REGION Network 4: Block description — Section 3.3 to 3.5
   // ▂▂▂▂▂▂▂▂▂▂▂▂▂▂▂▂▂▂▂▂▂▂▂▂▂▂▂▂▂▂▂▂▂▂▂▂▂▂▂▂▂▂▂▂
   // 3.3     Fault handling
   // 
   // 
   // There are five fault conditions, four are derived from position faults and one from an external 
   // fault signal:
   // 
   //  ――――――――――――――――――――――――――――――――――――――――――
   //  FAULT         DESCRIPTION                     LATCHING
   //  ――――――――――――――――――――――――――――――――――――――――――
   //  Failed to open      Valve failed to open in the specified               YES
   //             opening operation time
   // 
   //  Failed to close      Valve failed to close in the specified              YES
   //             closing operation time
   // 
   //  Failed while open   Valve suffered position failure while            YES
   //             in a static OPEN state
   // 
   //  Failed while closed   Valve suffered position failure while            YES
   //             in a static CLOSED state
   // 
   //  External fault        The EXT_FAULT signal is active                 NO
   //   ――――――――――――――――――――――――――――――――――――――――――
   // 
   // If any of the above faults are active, the valve will be deenergised (both the OPEN_CMD and 
   // CLOSE_CMD parameters will be set to 0) and the module will ignore all commands either 
   // automatic or manual and will ignore all interlock conditions.
   // 
   // Note:    If the maintain output option is activated (CONFIG_MAINT_OP = 1), the outputs will be 
   //      deenergised if a fault is present (both the OPEN_CMD and CLOSE_CMD parameters 
   //      will be set to 0).
   // 
   // 
   // 
   // ▁▁▁▁▁▁▁▁▁▁▁▁▁▁▁▁▁▁▁▁▁▁▁▁▁▁▁▁▁▁▁▁▁▁▁▁▁▁▁▁▁▁▁▁
   // 3.3.1    Position faults
   // 
   // 
   // All position faults (derived from position feedback signals) are latching fault conditions that  
   // require the operator to issue a reset command, this is usually via a faceplate available at the 
   // supervisory system (SCADA/HMI), but could also be via a hardwired 
   // (pushbutton) signal. 
   // 
   // The reset signal is specified within the DYNAMIC_DATA parameter UDT as follows:        
   // 
   //  DATA STRUCTURE    UT31101_Dy_DevValveBi
   //  ――――――――――――――――――――――――――――――――――――――――――
   //  SIGNAL         FUNCTION                TYPE     DETAILS
   //  ――――――――――――――――――――――――――――――――――――――――――
   //  mode_Reset        A reset pulse                Bool     1 = reset latched faults
   //            (active for one Controller cycle)            0 = no action
   //  ――――――――――――――――――――――――――――――――――――――――――
   // 
   // 
   // 
   // ▁▁▁▁▁▁▁▁▁▁▁▁▁▁▁▁▁▁▁▁▁▁▁▁▁▁▁▁▁▁▁▁▁▁▁▁▁▁▁▁▁▁▁▁
   // 3.3.2    Resetting position faults
   // 
   // 
   // If a position fault has occurred, and the fault is then reset, the appropriate opening or closing 
   // operation timer will be retriggered, allowing the valve time to achieve the required position.
   // 
   // 
   // 
   // ▁▁▁▁▁▁▁▁▁▁▁▁▁▁▁▁▁▁▁▁▁▁▁▁▁▁▁▁▁▁▁▁▁▁▁▁▁▁▁▁▁▁▁▁
   // 3.3.3    External fault
   // 
   // 
   // The external fault is an optional hardwired signal from the valve, it indicates that the device 
   // itself is registering that there is some problem. Such external fault signals are more commonly 
   // associated with motorised valves (equipped with thermal overload detectors), but may also be 
   // associated with pneumatic or hydraulic operated valves to indicate that the is a 
   // pneumatic/hydraulic system failure.
   // 
   // Such fault signals are generally indicated via a hardwired digital input to the Controller.
   // 
   // The external fault signal (if used) is passed to the module as the parameter: EXT_FAULT .
   // 
   // Any signal connected to the EXT_FAULT parameter must be active high (i.e. the signal must be 
   // set to 1 to indicate the fault condition is present). 
   // 
   // Where a failsafe response signal is used (active when set to 0) is used, it must be inverted at the 
   // EXT_FAULT parameter:
   // 
   // 
   //                         ┌─────────────
   //      ───────────────────┤ FC11101 
   //                         ├───────────────┤
   //           "V001_FAULT"               │               │
   //        ────┤╱├──────────┤ EXT_FAULT             │
   //                         │               
   //                         │               
   // 
   // 
   // If the EXT_FAULT signal is not required, the input should be set to _False  (similar to the safety 
   // and interlock signals that are not used, see § 3.4).
   // 
   // The EXT_FAULT signal is non-latching; it does not require a mode_Reset signal to clear the fault. 
   // The external fault will automatically reset whenever the EXT_FAULT signal is set to 0.
   // 
   // 
   // 
   // ▂▂▂▂▂▂▂▂▂▂▂▂▂▂▂▂▂▂▂▂▂▂▂▂▂▂▂▂▂▂▂▂▂▂▂▂▂▂▂▂▂▂▂▂
   // 3.4     Safety and interlocks
   // 
   // 
   // Safety and interlock signals are optional signals, passed as individual parameters to the module 
   // (in the same a manner as IO signals), all such signals are optional, a valve can have all, none or 
   // any combination of the signals.
   // 
   // Safety and interlock signals all act to override the normal operation of the valve (whether in 
   // automatic or manual mode) and force the valve to a particular state.
   // 
   // There is one safety signal and three interlock signals, each having its own formal module 
   // parameter:
   // 
   // 
   //  SAFETY SIGNAL
   //  ――――――――――――――――――――――――――――――――――――――――――
   //  PARAM        FUNCTION                   TYPE     DETAILS 
   //  ――――――――――――――――――――――――――――――――――――――――――
   //  E_STOP       Safety or emergency stop signals are         Bool     1 = E-stop active
   //          hardwired signals that remove power            0 = healthy
   //          required, set permanently to _False
   //  ――――――――――――――――――――――――――――――――――――――――――
   //  INTERLOCK SIGNALS
   //  ――――――――――――――――――――――――――――――――――――――――――
   //  PARAM        FUNCTION                   TYPE     DETAILS  
   //  ――――――――――――――――――――――――――――――――――――――――――
   //  TRIP       A latching interlock, it activates whenever a      Bool     1 = Trip active
   //          set of events are true and forces the devices        0 = healthy
   //          to a given state. It will not deactivate until the 
   //          triggering conditions are removed and a 
   //          reset signal has been given.
   // 
   //  INTERLOCK    A simple interlock that is active whenever a   Bool     1 = Interlock active
   //          set of conditions is true, it will force the            0 = healthy
   //          devices to a given state
   // 
   //  PERMISSIVE     Takes no action if a device is in a non-        Bool     1 = Permissive active
   //          permitted state, but once the device is in           0 = healthy
   //          that state will prevent a transition back to 
   //          the non-permitted state.
   //  ――――――――――――――――――――――――――――――――――――――――――
   // 
   // 
   // Each safety and interlock signal has its own configuration signal that must be used to formally 
   // disable the parameter if the signal is not required, these are all within the STATIC_DATA parameter 
   // UDT (UT11101_St_DevValveBi) as follows:
   // 
   // 
   //  DATA STRUCTURE    UT11101_St_DevValveBi
   //  ――――――――――――――――――――――――――――――――――――――――――
   //  SIGNAL        FUNCTION              TYPE     DETAILS
   //  ――――――――――――――――――――――――――――――――――――――――――
   //  CONFIG_ESTOP_DIS    Disables the safety signal.        Bool     1 = E_STOP disabled
   //              If set to 1, any signal on the          0 = E_STOP enabled
   //              E_STOP parameter will be 
   //              ignored.
   // 
   //  CONFIG_TRIP_DIS      Disables the trip interlock signal.   Bool     1 = TRIP disabled
   //              If set to 1, any signal on the          0 = TRIP enabled
   //              TRIP parameter will be 
   //              ignored.
   // 
   //  CONFIG_ILOCK_DIS     Disables the interlock signal.    Bool     1 = INTERLOCK disabled
   //              If set to 1, any signal on the          0 = INTERLOCK enabled
   //              INTERLOCK parameter will be 
   //              ignored.
   // 
   //  CONFIG_PERM_DIS   Disables the permissive interlock  Bool     1 = PERMISSIVE disabled
   //              signal. If set to 1, any signal on the       0 = PERMISSIVE enabled
   //              TRIP parameter will be 
   //              ignored.
   //  ――――――――――――――――――――――――――――――――――――――――――
   // 
   // The disable signals are used to formally configure the valve, they allow any supervisory system to 
   // know the correct configuration of the valve and display information accordingly.
   // 
   // 
   // 
   // ▁▁▁▁▁▁▁▁▁▁▁▁▁▁▁▁▁▁▁▁▁▁▁▁▁▁▁▁▁▁▁▁▁▁▁▁▁▁▁▁▁▁▁▁
   // 3.4.1    Safety signal operation
   // 
   // 
   // Safety or emergency stop signals are hardwired signals that remove power from a device forcing 
   // it to a safe state. Such signals act independently of the software (the pressing of an emergency 
   // stop button will physically remove power from the affected devices).
   // 
   // The emergency stop signal is passed to the module as the parameter E_STOP; it informs the 
   // module that the safety signal has been activated and allows the module to adjust the state of 
   // the valve to follow the emergency stop conditions.
   // 
   // When the emergency stop signal is removed, the valve will resume the requested state (with the 
   // appropriate operation timer).
   // 
   // Under emergency stop conditions the valve is always deenergised (both physically by the 
   // hardware and within the software via the actions of this module), both the OPEN_CMD and 
   // CLOSE_CMD outputs set to zero (OPEN_CMD = 0 and CLOSE_CMD = 0).
   // 
   // The emergency stop signal is absolute and will override any other demand made of the valve. 
   // There is no mechanism for bypassing this form of safety signal.
   // 
   // 
   // 
   // ▁▁▁▁▁▁▁▁▁▁▁▁▁▁▁▁▁▁▁▁▁▁▁▁▁▁▁▁▁▁▁▁▁▁▁▁▁▁▁▁▁▁▁▁
   // Safety signal operation when valve is changing state (recovery time)
   // 
   // 
   // In the case of a bistable valve, the removing of the power under emergency stop conditions, 
   // simply deenergises both outputs leaving the valve in its current state: if the valve were already 
   // open, it would remain open, similarly if the valve were closed, it would remain closed.
   // 
   // Additionally, if the valve were in the process of changing state (either opening or closing) when 
   // the emergency stop occurred, the same thing happens, both outputs are deenergised and the 
   // valve simply stops where it is in mid-transition (i.e. in some indeterminate, intermediate state 
   // between open and closed). 
   // 
   // To accommodate this condition, the active operation timer will simply pause at its current 
   // elapsed value (the value reached when the emergency stop activated) and the valve will 
   // remain in either the opening or closing state; i.e. status_Opening or status_Closing will remain 
   // active until the emergency stop condition is removed.
   // 
   // Under these conditions (an emergency stop while changing state), the removal of the 
   // emergency stop tiggers a recovery timer, this is used to delay the restarting of the operation 
   // timer (or the run-on timer if it is active), the recover timer is used to allow the physical aspects 
   // of the valve itself to reset and resume operation (e.g. to allow the valve to power-up and the 
   // motor to ramp to the correct speed &c.), this recovery time is configurable.
   // 
   // Note:    The recovery timer will also run when the emergency stop condition is removed 
   //      even if the valve is in a defined position, under these circumstances, the operation 
   //      timer will again be delayed until the recovery timer is complete (this avoids a 
   //      situation where the valve is required to change state immediately after an estop 
   //      while the valve motor is still recovering — again it effectively extends the operation 
   //      timer sufficiently to allow the valve to recover).
   // 
   // The recovery time preset is specified in the STATIC_DATA parameter 
   // UDT (UT11101_St_DevValveBi) as follows. It is the same irrespective of whether the valve was 
   // opening or closing.
   // 
   // 
   //  DATA STRUCTURE    UT11101_St_DevValveBi
   //  ――――――――――――――――――――――――――――――――――――――――――
   //  SIGNAL        FUNCTION              TYPE     DETAILS
   //  ――――――――――――――――――――――――――――――――――――――――――
   //  TIME_RECOVERY       Recovery delay time, delays the     Real     Seconds
   //              restarting of the operation time 
   //              if an E stop occurred while 
   //              changing state
   //  ――――――――――――――――――――――――――――――――――――――――――
   // 
   // 
   // If the recovery timer is active, the elapsed (counting down) time is stored within the 
   // DYNAMIC_DATA parameter UDT (UT31101_Dy_DevValveBi) as follows:
   // 
   // 
   //  DATA STRUCTURE    UT31101_Dy_DevValveBi
   //  ――――――――――――――――――――――――――――――――――――――――――
   //  SIGNAL        FUNCTION              TYPE     DETAILS
   //  ――――――――――――――――――――――――――――――――――――――――――
   //  actual_Recovery_Timer    Actual (elapsed) value of     Real     Seconds
   //              the recovery timer  
   //  ――――――――――――――――――――――――――――――――――――――――――
   // 
   // 
   // Again, the recovery timer counts down from the TIME_RECOVERY value to zero, at which point, the 
   // operation timer will restart from the elapsed time.
   // 
   // Note:    During the recovery period, the appropriate OPEN_CMD or CLOSE_CMD output will 
   //      reactivate (depending on whether the valve was originally opening or closing).
   // 
   // 
   // 
   // ▁▁▁▁▁▁▁▁▁▁▁▁▁▁▁▁▁▁▁▁▁▁▁▁▁▁▁▁▁▁▁▁▁▁▁▁▁▁▁▁▁▁▁▁
   // Typical usage of the E_STOP parameter
   // 
   // 
   // Any safety signal connected to the E_STOP parameter must be active high (i.e. the signal must be 
   // set to 1 to activate the safety signal response). It is often the case, where hardwired emergency 
   // stop signals are used, that the emergency stop condition is activated by the absence of a signal 
   // (a failsafe response) rather than the application of a signal. The module can accommodate this 
   // sense of signal by inverting the E_STOP input:
   // 
   // 
   //                         ┌─────────────
   //      ───────────────────┤ FC11101 
   //                         ├───────────────┤
   //           "ZONEA_ESTOP"              │               │
   //        ────┤╱├──────────┤ E_STOP             │
   //                         │               
   //                         │               
   // 
   // 
   // If no safety signal is used, the parameter is set to the _False tag (note, also that the configuration 
   // signal CONFIG_ESTOP_DIS should also be set to 1):
   // 
   // 
   //                         ┌─────────────
   //      ───────────────────┤ FC11101 
   //                         ├───────────────┤
   //                         │               │
   //                      _False ──┤ E_STOP             │
   //                         │               
   //                         │    
   // 
   // 
   // 
   // ▁▁▁▁▁▁▁▁▁▁▁▁▁▁▁▁▁▁▁▁▁▁▁▁▁▁▁▁▁▁▁▁▁▁▁▁▁▁▁▁▁▁▁▁
   // 3.4.2    Interlock signals
   // 
   // 
   // Interlock signals are a more flexible mechanism for overriding the requested position of the valve. 
   // Interlock signals can be both hardware driven (similar to a safety signal) or can be purely software 
   // derived (unlike a safety signal).
   // 
   // Software derived interlock signals can accommodate more complex and more flexible 
   // arrangements, it would for example, be possible to disable a software derived interlock if the 
   // process were undergoing some particular function, such as cleaning &c.
   // 
   // There are three different types of interlock arrangements:
   // 
   // There are three types of interlock signal:
   // 
   //    1.  INTERLOCK
   //      A simple interlock that is active whenever a set of conditions is true, it will force any 
   //      associated devices to a given safe state.
   // 
   //    2.  PERMISSIVE
   //      Takes no action if a device is in a non-safe state, but once the device is in a safe 
   //      state will prevent a transition to a non-safe state (i.e. will not force a valve to close, 
   //      but once it is closed, will prevent it from re-opening).
   // 
   //    3.  TRIP
   //      A latching interlock, it activates whenever a set of events are true (like an interlock), 
   //      but will not deactivate until the triggering conditions are removed and a reset signal 
   //      has been given (effectively a latching interlock), it will force any associated devices 
   //      to a given safe state.
   // 
   // For any type of interlock, the specified interlock state (or permitted state) can be either open or 
   // closed irrespective of the type of valve (normally open or normally closed); unlike the safety signal, 
   // it does not have to be the deenergised state of the valve.
   // 
   // That said, the most common interlock state is the deenergised state of the valve; i.e. the failsafe 
   // position of the valve.
   // 
   // 
   // 
   // ▁▁▁▁▁▁▁▁▁▁▁▁▁▁▁▁▁▁▁▁▁▁▁▁▁▁▁▁▁▁▁▁▁▁▁▁▁▁▁▁▁▁▁▁
   // Typical usage of interlock signals
   // 
   // 
   // Each type of interlock is passed as its own parameter: TRIP, INTERLOCK or PERMISSIVE. Like the 
   // safety signal (E_STOP), each parameter is active high (i.e. the signal must be set to 1 to activate 
   // the associated interlock signal response). 
   // 
   // Again, it is often the case, where hardwired interlock signals are used, that the condition is 
   // activated by the absence of a signal (i.e. a failsafe response) rather than the application of a 
   // signal. The module can accommodate this sense of signal by inverting the relevant input:
   // 
   // 
   //                         ┌─────────────
   //      ───────────────────┤ FC11101 
   //                         ├───────────────┤
   //        "DB23102_Dy_Perm.V001"     │               │
   //        ────┤╱├──────────┤ PERMISSIVE           │
   //                         │               
   // 
   // If a particular interlock signal is not used, the parameter is set to the _False tag (note also: that 
   // the appropriate configuration signal should also be set to 1: CONFIG_TRIP_DIS, CONFIG_ILOCK_DIS 
   // or CONFIG_PERM_DIS).
   // 
   //                         ┌─────────────
   //      ───────────────────┤ FC11101 
   //                         ├───────────────┤
   //                         │               │
   //                      _False ──┤ TRIP                    │
   //                         │               
   //                         │  
   // 
   // 
   // 
   // ▁▁▁▁▁▁▁▁▁▁▁▁▁▁▁▁▁▁▁▁▁▁▁▁▁▁▁▁▁▁▁▁▁▁▁▁▁▁▁▁▁▁▁▁
   // Configuring the interlock signals
   // 
   // 
   // The state adopted by the valve when a particular interlock is active (TRIP or INTERLOCK) or the 
   // permitted state of the valve (PERMISSIVE) are set individually for each type of interlock signal. 
   // These configuration signals are stored within the STATIC_DATA parameter UDT as follows:
   // 
   // 
   //  DATA STRUCTURE    UT11101_St_DevValveBi
   // 
   //  ――――――――――――――――――――――――――――――――――――――――――
   //  SIGNAL        FUNCTION              TYPE     DETAILS
   //  ――――――――――――――――――――――――――――――――――――――――――
   //  CONFIG_TRIP_OP_CL   The required state of a valve if     Bool     1 = valve will open
   //              the TRIP signal is active            0 = valve will close
   // 
   //  CONFIG_ILOCK_OP_CL  The required state of a valve if     Bool     1 = valve will open
   //              the INTERLOCK signal is active         0 = valve will close
   // 
   //  CONFIG_PERM_OP_CL  The permitted state of a valve if   Bool     1 = valve may open
   //              the PERMISSIVE signal is active          0 = valve may close
   //  ――――――――――――――――――――――――――――――――――――――――――
   // 
   // For example, if CONFIG_ILOCK_OP_CL is set to 1, the valve will open whenever the INTERLOCK 
   // signal is active (set to 1), this will override any automatic or manual requirement for the valve 
   // (but will not override a safety signal, see below). If CONFIG_ILOCK_OP_CL were set to 0, the 
   // valve would close whenever the INTERLOCK signal was active.
   // 
   // The TRIP signal behaves in exactly the same way as the INTERLOCK signal, but uses 
   // CONFIG_TRIP_OP_CL to set the tripped state of the valve.
   // 
   // Although the TRIP signal requires a reset signal to disengage the interlock conditions, this is 
   // handled by the trip logic itself (usually handled by the trip application modules: FC23200) and 
   // not via this module; simply deactivating the TRIP signal removes the trip state from the valve 
   // and allows it to operate normally.
   // 
   // The PERMISSIVE signal operates in a different way, if CONFIG_PERM_OP_CL were set to 1 
   // (valve is permitted to open), and the valve was currently closed under automatic control when 
   // the PERMISSIVE signal became active, nothing would happen to the valve (it would remain 
   // closed), if the valve then subsequently opened under automatic control, the PERMISSIVE signal
   //  would allow the valve to do so (the valve permitted state is open). However, any attempt by 
   // the automatic system to re-close the valve would not be allowed by the PERMISSIVE signal.
   // 
   // Conversely, if CONFIG_PERM_OP_CL were set to 0 (valve is permitted to close), and the valve 
   // was currently open under automatic control when the PERMISSIVE signal became active, 
   // nothing would happen to the valve (it would remain open), if the valve then subsequently 
   // closed under automatic control, the PERMISSIVE signal would allow the valve to do so (the 
   // valve permitted state is close). However, any attempt by the automatic system to re-open 
   // the valve would not be allowed by the PERMISSIVE signal.
   // 
   // Note:    Where multiple interlock signals are used, it is possible for the different interlocks 
   //      to apply different states to the valve, for example an active TRIP could close 
   //      the valve and an active INTERLOCK open it. Such conflicts are managed by the 
   //      different priorities applied to the interlock signals (see § 3.5).  
   // 
   // 
   // 
   // ▁▁▁▁▁▁▁▁▁▁▁▁▁▁▁▁▁▁▁▁▁▁▁▁▁▁▁▁▁▁▁▁▁▁▁▁▁▁▁▁▁▁▁▁
   // Bypassing interlocks
   // 
   // 
   // Unlike safety signals, all interlock signals can be overridden (or bypassed). The bypass signal is a 
   // single signal that, if active, overrides and deactivates any TRIP, INTERLOCK or PERMISSIVE signal 
   // that may have been activated.
   // 
   // The bypass signal is specified within the DYNAMIC_DATA parameter UDT as follows:
   // 
   // 
   //  DATA STRUCTURE    UT31101_Dy_DevValveBi
   //  ――――――――――――――――――――――――――――――――――――――――――
   //  SIGNAL         FUNCTION                TYPE     DETAILS
   //  ――――――――――――――――――――――――――――――――――――――――――
   //  mode_BypassOn   Activates bypass mode, if active, any    Bool     1 = bypass mode on
   //            TRIP, INTERLOCK or PERMISSIVE signal          0 = bypass mode off
   //            will be ignored
   //  ――――――――――――――――――――――――――――――――――――――――――
   // 
   // 
   // Bypass mode is a manual operation, generally activated by the operator via a faceplate 
   // available at the supervisory system (SCADA/HMI), or via some hardwired signal, such as 
   // a key-switch.
   // 
   // It is possible to configure the module such that bypass mode is permanently disabled, this uses 
   // the following STATIC_DATA parameter:
   // 
   // 
   //  DATA STRUCTURE    UT11101_St_DevValveBi
   //  ――――――――――――――――――――――――――――――――――――――――――
   //  SIGNAL       FUNCTION                TYPE     DETAILS
   //  ――――――――――――――――――――――――――――――――――――――――――
   //  CONFIG_BYPASS_DIS    Prevents bypass mode being      Bool     1 = no bypass mode
   //             activated under all circumstances         0 = bypass permitted
   //  ――――――――――――――――――――――――――――――――――――――――――
   //   
   // If bypass mode is disabled (configuration signal CONFIG_BYPASS_DIS is set to 1), then the bypass 
   // mode cannot be turned on under any circumstances, the option will be greyed out on the 
   // supervisory system faceplate and the module will constantly reset the mode_BypassOn signal.
   // 
   // Note:    Safety (E_STOP) signals cannot be bypassed.  
   // 
   //      Similarly, if an interlock signal has a hardwired component (that will override any 
   //      software actions), it also must not be bypassed.
   // 
   // 
   // 
   // ▂▂▂▂▂▂▂▂▂▂▂▂▂▂▂▂▂▂▂▂▂▂▂▂▂▂▂▂▂▂▂▂▂▂▂▂▂▂▂▂▂▂▂▂
   // 3.5     Priority of operation
   // 
   // 
   // The valve is normally controlled by either the automatic system or by manual (operator) control; 
   // however, this operation can be overridden by the various safety and interlock conditions 
   // that can apply to the valve. Each of these operations is assigned a priority and if more than one 
   // is active at the same time, the one with the highest priority will take precedence.
   // 
   // The priorities for the various operations is as follows:
   // 
   // 
   //  ――――――――――――――――――――――――――――――――――――――――――
   //  SIGNAL TYPE       PRIORITY   ASSIGNED VALUE       CAN BE BYPASSED
   //  ――――――――――――――――――――――――――――――――――――――――――
   //  Emergency Stop        High        40                NO
   //  Trip            ↑           30             YES
   //  Interlock            ↑           20             YES
   //  Permissive          ↑           10             YES
   //  Auto/manual control    Low         00                NO
   //  ――――――――――――――――――――――――――――――――――――――――――
   //  High priority signal take precedence over lower priority signals.
   // 
   // Thus, if both the TRIP signal, the INTERLOCK signal and automatic control signal were all active at 
   // the same time, the module will respond only to the TRIP signal (with the higher priority) and will 
   // react accordingly.
END_REGION

REGION Network 5: Block description — Section 3.6 to 4
   // ▂▂▂▂▂▂▂▂▂▂▂▂▂▂▂▂▂▂▂▂▂▂▂▂▂▂▂▂▂▂▂▂▂▂▂▂▂▂▂▂▂▂▂▂
   // 3.6     Operating modes
   // 
   // 
   // This module FC11101_StdDevValveBi supports various operating modes:
   // 
   //    •   Automatic/manual mode
   // 
   //    •   Interlock bypass mode
   // 
   //    •   Simulation mode
   // 
   //    •   Remote/local mode
   // 
   //    •   Faceplate disabled mode
   // 
   // Examining these in turn:   
   // 
   // 
   // 
   // ▁▁▁▁▁▁▁▁▁▁▁▁▁▁▁▁▁▁▁▁▁▁▁▁▁▁▁▁▁▁▁▁▁▁▁▁▁▁▁▁▁▁▁▁
   // 3.6.1    Automatic and manual modes
   // 
   // 
   // Under normal operation, the valve is in automatic mode and is controlled directly by the 
   // Controller software (usually, sequential or continuous logic); however, it is possible for the 
   // operator to take direct control of the valve by switching it to manual mode.
   // 
   // If manual mode is active, the valve will open and close directly at the command of the operator 
   // and will ignore any automatic mode open and close requests.
   // 
   // If the valve is operating under automatic mode, the manual open/close request follows that of 
   // the automatic mode; this ensures that the valve remains in the same state when initially 
   // switched from automatic mode to manual mode, referred to as bumpless transfer. This approach 
   // minimises any disturbance to the process should the valve be inadvertently switched to manual 
   // mode.
   // 
   // The following data points are associated with automatic/manual mode:
   // 
   //  DATA STRUCTURE    UT11101_St_DevValveBi
   //  ――――――――――――――――――――――――――――――――――――――――――
   //  SIGNAL         FUNCTION               TYPE     DETAILS
   //  ――――――――――――――――――――――――――――――――――――――――――
   //  CONFIG_MAN_DIS     Prevents manual mode being       Bool  1 = no manual mode
   //            activated under all circumstances            0 = manual permitted
   //  ――――――――――――――――――――――――――――――――――――――――――
   // 
   //  DATA STRUCTURE    UT31101_Dy_DevValveBi
   //  ――――――――――――――――――――――――――――――――――――――――――
   //  SIGNAL         FUNCTION               TYPE     DETAILS
   //  ――――――――――――――――――――――――――――――――――――――――――
   //  Mode_AutMan     Identifies the operating mode of     Bool  1 = automatic mode
   //            the valve.                   0 = manual mode
   // 
   //  ctrl_Aut_OpenClose Causes the valve to open and close     Bool  1 = open the valve
   //            if automatic mode is active            0 = close the valve
   // 
   //  ctrl_Man_OpenClose  Causes the valve to open and close     Bool  1 = open the valve
   //            if manual mode is active             0 = close the valve
   // 
   //  status_Aut      The valve is in automatic mode      Bool  1 = auto mode
   //                                  0 = no in auto
   // 
   //  status_Man       The valve is in manual mode     Bool  1 = manual mode
   //                                  0 = no in manual
   //  ――――――――――――――――――――――――――――――――――――――――――
   // 
   // Manual mode can only be activated by the operator via a faceplate available at the supervisory 
   // system (SCADA/HMI).
   // 
   // If the manual mode is disabled (CONFIG_MAN_DIS = 1), then manual mode cannot be turned on 
   // under any circumstances, the option will be greyed out on the supervisory system faceplate and 
   // the valve will be permanently set to automatic mode (Mode_AutMan = 1).
   // 
   // 
   // 
   // ▁▁▁▁▁▁▁▁▁▁▁▁▁▁▁▁▁▁▁▁▁▁▁▁▁▁▁▁▁▁▁▁▁▁▁▁▁▁▁▁▁▁▁▁
   // 3.6.2    Interlock bypass mode
   // 
   // 
   // All interlock signals (TRIP, INTERLOCK or PERMISSIVE) can be overridden (bypassed). The bypass 
   // signal is a single signal that, if active, overrides and deactivates any TRIP, INTERLOCK or 
   // PERMISSIVE signal that may have been activated.
   // 
   // It is possible to permanently disable the bypass mode for any given valve (preventing the 
   // operator from activating it).
   // 
   // The following data points are associated with the bypass mode:
   // 
   //  DATA STRUCTURE    UT11101_St_DevValveBi
   //  ――――――――――――――――――――――――――――――――――――――――――
   //  SIGNAL       FUNCTION                TYPE     DETAILS
   //  ――――――――――――――――――――――――――――――――――――――――――
   //  CONFIG_BYPASS_DIS    Prevents bypass mode being      Bool     1 = no bypass mode
   //             activated under all circumstances         0 = bypass permitted
   //  ――――――――――――――――――――――――――――――――――――――――――
   // 
   //  DATA STRUCTURE    UT31101_Dy_DevValveBi
   //  ――――――――――――――――――――――――――――――――――――――――――
   //  SIGNAL         FUNCTION                TYPE     DETAILS
   //  ――――――――――――――――――――――――――――――――――――――――――
   //  mode_BypassOn   Activates bypass mode, if active, any    Bool     1 = bypass mode on
   //            TRIP, INTERLOCK or PERMISSIVE signal          0 = bypass mode off
   //            will be ignored
   // 
   //  status_BypassOn   Status indication, shows if bypass      Bool     1 = bypass active
   //            mode is active                 0 = bypass inactive
   //  ――――――――――――――――――――――――――――――――――――――――――
   // 
   // Bypass mode can only be activated by the operator usually via a faceplate available at the 
   // supervisory system (SCADA/HMI), alternatively it may be via some form of hardwired signal such 
   // as a key-switch &c. 
   // 
   // If bypass mode is disabled (configuration signal CONFIG_BYPASS_DIS is set to 1), then the bypass 
   // mode cannot be turned on under any circumstances, the option will be greyed out on the 
   // supervisory system faceplate and the module will constantly reset the mode_BypassOn signal.  
   // 
   // 
   // 
   // ▁▁▁▁▁▁▁▁▁▁▁▁▁▁▁▁▁▁▁▁▁▁▁▁▁▁▁▁▁▁▁▁▁▁▁▁▁▁▁▁▁▁▁▁
   // 3.6.3    Simulation mode
   // 
   // 
   // The module can be switched to a simulation mode, in which the position feedback for the valve 
   // is replaced by simulated signals specified by the operator. 
   // 
   // Simulation mode is generally used during testing, but can also be applied in a process 
   // environment if a fault condition is detected; this scenario allows the plant to continue operating 
   // (albeit under some degree of manual control) until the valve is repaired or replaced.
   // 
   // The following data points are associated with the simulation mode:
   // 
   //  DATA STRUCTURE    UT11101_St_DevValveBi
   //  ――――――――――――――――――――――――――――――――――――――――――
   //  SIGNAL       FUNCTION                TYPE     DETAILS
   //  ――――――――――――――――――――――――――――――――――――――――――
   //  CONFIG_SIM_DIS     Prevents simulation mode being     Bool     1 = no sim mode
   //             activated under all circumstances         0 = sim permitted
   //  ――――――――――――――――――――――――――――――――――――――――――
   // 
   //  DATA STRUCTURE    UT31101_Dy_DevValveBi
   //  ――――――――――――――――――――――――――――――――――――――――――
   //  SIGNAL         FUNCTION                TYPE     DETAILS
   //  ――――――――――――――――――――――――――――――――――――――――――
   //  mode_SimOn      Activates simulation mode, if active, the   Bool     1 = sim mode on
   //            position feedback will be specified by         0 = sim mode off
   //            mode_SimValue      
   //  mode_SimValue    Specifies the type of simulated position     Int     0 = no feedback
   //            feedback in use                  1 = permanently open
   //                                      2 = permanently closed
   //                                      3 = follow demand
   // 
   //  status_SimOn     Status indication, shows if simulation     Bool     1 = sim active
   //            mode is active                 0 = sim inactive
   //  ――――――――――――――――――――――――――――――――――――――――――
   // 
   // Simulation mode can only be activated by the operator via a faceplate available at the 
   // supervisory system (SCADA/HMI).
   // 
   // If simulation mode is activated, the position feedback for the valve is forced to one of four 
   // states specified by the mode_SimValue variable (this is an enumerated variable):
   // 
   //  ――――――――――――――――――――――――――――――――――――――――――
   //  mode_SimValue  DESCRIPTION               FBK_OPEN FBK_CLOSED
   //  ――――――――――――――――――――――――――――――――――――――――――
   //      0        Permanently disables all position feedback    0     0
   //             (irrespective of any valve position)
   // 
   //      1        Permanently sets valve position to open         1     0
   //             (irrespective of any valve position)
   // 
   //      2        Permanently sets valve position to closed      0     1
   //             (irrespective of any valve position)
   // 
   //      3        Position feedback follows the requested        1/0    0/1
   //             state of the valve              (if valve is open/closed)
   //  ――――――――――――――――――――――――――――――――――――――――――
   // 
   // The mode_SimValue is restricted to the range 0-3.
   // 
   // If simulation mode is disabled (configuration signal CONFIG_SIM_DIS is set to 1), then the 
   // simulation mode cannot be turned on under any circumstances, the option will be greyed out on 
   // the supervisory system faceplate and the module will constantly reset the mode_SimOn signal.
   // 
   // If simulation mode is permitted (CONFIG_SIM_DIS = 0), then setting mode_SimOn to 1 will activate 
   // simulation mode and the any position feedback signals (connected to FBK_OPEN and 
   // FBK_CLOSED) will be overridden according to the value stored in mode_SimValue (see Table above).
   // 
   // The operator can set and adjust the simulation value (mode_SimValue) from the instrument 
   // faceplate on the supervisory system. The simulation value can be adjusted at any time by the 
   // operator (even if simulation mode has not been activated), but will not be applied until 
   // simulation mode is turned on (mode_SimOn = 1). 
   // 
   // If simulation mode is completely disabled (CONFIG_SIM_DIS is set to 1) then the operator will not 
   // be able to adjust the simulated value (mode_SimValue will be greyed out on the faceplate).
   // 
   // 
   // 
   // ▁▁▁▁▁▁▁▁▁▁▁▁▁▁▁▁▁▁▁▁▁▁▁▁▁▁▁▁▁▁▁▁▁▁▁▁▁▁▁▁▁▁▁▁
   // A note on the follow demand simulation mode
   // 
   // The follow demand simulation mode for a bistable valve is subtly different to that of an isolating 
   // valve (cf. FC11001). With the isolating valve, the follow demand simulation mode changes the 
   // state of the valve instantly when the demand changes (it does not wait for any operation time), 
   // this is an acceptable response for an isolating valve which maintains its output signal in the 
   // required state whilever the demand is present.
   // 
   // With a bistable valve, the outputs (generally) deenergise when the correct state is reached. Thus 
   // the follow demand simulation mode for a bistable valve will switch to the required state just prior 
   // to the expiration of the operation timer. This allows the output signals to be maintained for the 
   // maximum length of time ensuring the valve has actually reached the required state.
   // 
   // In practice, the simulated state signals will be generated approximately 200ms before the 
   // operation timer would expire.
   // 
   // 
   // 
   // ▁▁▁▁▁▁▁▁▁▁▁▁▁▁▁▁▁▁▁▁▁▁▁▁▁▁▁▁▁▁▁▁▁▁▁▁▁▁▁▁▁▁▁▁
   // 3.6.4     Remote/local mode
   // 
   // Remote and local operating modes refer to the supervisory system that has control of the 
   // device (i.e. which system can write to the device and change the operating mode of the 
   // device). 
   // 
   // This type of mode is usual present where a plant has a remote central control location (a control 
   // room) that normally controls the device (remote control), but also has a field panel with a local 
   // HMI that an operator in the field can select to take over control of the device (local control) for 
   // maintenance purposes.
   // 
   // The modes are as follows (and are mutually exclusive, only one will be active):
   // 
   //    Remote        Only the remote system in the control room can 
   //                 control the device
   // 
   //    Local            A local system has taken control of the device and the remote 
   //                 system can no longer issue commands to it
   // 
   //    Remote/local disabled   The system does not use remote/local modes and any 
   //      (ALL mode)     supervisory system can issue commands to the device 
   //  
   // Remote/local control is generally handled by the supervisory systems themselves; however, the 
   // supervisory systems need a storage area per device to record which mode that device is in, local 
   // control is often activated by a panel key-switch, that changes the state of several devices from 
   // remote to local (usually all the devices controlled by the local panel).
   // 
   // The module simply identifies the remote/local mode from the mode signals and configuration 
   // signals provided to the module.
   // 
   // For systems that do not use remote/local modes (any supervisory system can control the device, 
   // or control is determined by operator privileges), the remote/local modes can be disabled 
   // (CONFIG_RL_EN is set to zero) and the device is effectively in ALL mode (any system can 
   // control the device).
   // 
   // If remote/local operation is in use, the supervisory system that does not have control will still 
   // display all the information from the device, but will not be able to control the device (it could not 
   // for example, activate simulation mode) and all control function (faceplate functions) will be 
   // greyed out.
   // 
   // The following signals are associated with remote/local/all modes:
   // 
   //  DATA STRUCTURE    UT11101_St_DevValveBi
   //  ――――――――――――――――――――――――――――――――――――――――――
   //  SIGNAL           FUNCTION            TYPE   DETAILS
   //  ――――――――――――――――――――――――――――――――――――――――――
   //  CONFIG_RL_EN      Allows Remote and Local      Bool    1 = Remote/local selected
   //                 modes to be selected        0 = All mode is active
   // 
   //  DATA STRUCTURE    UT31101_Dy_DevValveBi
   //  ――――――――――――――――――――――――――――――――――――――――――
   //  SIGNAL           FUNCTION            TYPE   DETAILS
   //  ――――――――――――――――――――――――――――――――――――――――――
   //  mode_RemoteOn       Activates remote mode     Bool    1 = remote mode on, 
   //                 CONFIG_RL_EN must = 1       0 = remote mode off
   // 
   //  mode_LocalOn     Activates local mode          Bool    1 = local mode on, 
   //                 CONFIG_RL_EN must = 1       0 = remote mode off
   // 
   //  status_RemoteOn      Status remote mode on     Bool    1 = remote mode on, 
   //                               0 = remote mode off
   // 
   //  status_LocalOn       Status local mode on      Bool 1 = local mode on, 
   //                               0 = local mode off
   // 
   //  status_RLOff       Status ALL mode is on = 0    Bool 1 = ALL mode on, 
   //                               0 = ALL mode off
   //  ――――――――――――――――――――――――――――――――――――――――――
   //  Block remote/local signals 
   // 
   // By default, remote/local is disabled — ALL mode is selected (CONFIG_RL_EN = 0).
   // 
   // 
   // 
   // 
   // ▁▁▁▁▁▁▁▁▁▁▁▁▁▁▁▁▁▁▁▁▁▁▁▁▁▁▁▁▁▁▁▁▁▁▁▁▁▁▁▁▁▁▁▁
   // 3.6.5     Faceplate disable mode
   // 
   // It is possible to disable the supervisory system faceplate from within the module, the 
   // configuration signal:
   // 
   // 
   //  ――――――――――――――――――――――――――――――――――――――――――
   //  SIGNAL           FUNCTION            TYPE   DETAILS
   //  ――――――――――――――――――――――――――――――――――――――――――
   //  CONFIG_FP_DIS        Disable the supervisory      Bool    1 = Faceplate disabled
   //                 system faceplate           0 = normal
   //  ――――――――――――――――――――――――――――――――――――――――――
   // 
   // If the faceplate is disabled (CONFIG_FP_DIS = 1), the supervisory system must not allow the 
   // device faceplate to be opened (normally achieved by clicking the block icon or device symbol), 
   // this in turn prevents the operator from affecting the device in anyway, it would not, for example, 
   // be possible to put the device into simulation mode.
   // 
   // Similarly, if the faceplate is disabled, the operator will not have access to the mode_Reset signal, 
   // meaning that alternative reset mechanisms must be in place (such as a hardwired pushbutton 
   // for example).
   // 
   //                ━━━   ⬙⬙⬙⬙⬙⬙   ━━━
   // 
   // 
   // 
   // ▄▄▄▄▄▄▄▄▄▄▄▄▄▄▄▄▄▄▄▄▄▄▄▄▄▄▄▄▄▄▄▄▄▄▄▄▄▄▄▄▄▄▄▄
   // 4.     Supervisory system interface
   // 
   // 
   // See the online documentation for this block — select the block in the project tree and press:
   //      SHIFT + F1 or follow the link: https://psop.uk/pal-smds-fc11101-p 
   // 
   // An explanation of the block icons and faceplates available to the supervisory system for this 
   // module is given in section 4 of the SMDS document [Ref. 011].
   // 
   // A downloadable copy of the SMDS (and all other project documentation) is available here:
   // 
   //      https://practicalseries.com/2001-pal/21-project/01-00-docs.html
   // 
   // For this module, the document number is: PS2001-5-2312-fc11101
   // 
   //                ━━━   ⬙⬙⬙⬙⬙⬙   ━━━
END_REGION

REGION Network 6: Block description — Sections 5 to 11
   // ▄▄▄▄▄▄▄▄▄▄▄▄▄▄▄▄▄▄▄▄▄▄▄▄▄▄▄▄▄▄▄▄▄▄▄▄▄▄▄▄▄▄▄▄
   // 5.     PARAMETERS
   // 
   // 
   // The following parameters are associated with the block:
   // 
   //  
   //  ――――――――――――――――――――――――――――――――――――――――――
   //  PARAM         FUNCTION                    TYPE      IN-OUT 
   //  ――――――――――――――――――――――――――――――――――――――――――
   //  SYS_SIGNALS      Common system signals              UT21000    In
   //           logic and timing signals for parametric access
   // 
   //  FBK_OPEN     Optional open state positive feedback        Bool      In
   //           (1 = open, 0 = not open) If not required, set 
   //           permanently to _False
   // 
   //  FBK_CLOSED    Optional closed state positive feedback        Bool      In
   //           (1 = closed 0 = not closed) If not required, set 
   //           permanently to _False
   // 
   //  EXT_FAULT     Optional external fault signal for the device     Bool      In
   //           (1 = fault, 0 = healthy). If not required, set 
   //           permanently to _False
   // 
   //  E_STOP        Optional emergency stop (safety) signal        Bool      In
   //           (1 = emergency stop active, 0 = healthy) If not 
   //           required, set permanently to _False
   // 
   //  TRIP        Optional trip signal                  Bool      In
   //           (1 = trip condition active, 0 = healthy) If not 
   //           required, set permanently to _False
   // 
   //  INTERLOCK     Optional interlock signal               Bool      In
   //           (1 = interlock condition active, 0 = healthy) If 
   //           not required, set permanently to _False
   // 
   //  PERMISSIVE      Optional permissive signal             Bool      In
   //           (1 = permissive condition active, 0 = healthy) 
   //           If not required, set permanently to _False
   // 
   //  STATIC_DATA     Data structure that holds the configuration data     UT11101    In
   //           for the device (limit switch, timer presets 
   //           and interlock configuration &c.)
   // 
   //  DYNAMIC_DATA      Data structure that holds the live data for the       UT31101    InOut
   //           device (its mode, status, messages and 
   //           other dynamic information)
   // 
   //  OPEN_CMD       Output to drive the valve to an open state    Bool      Out
   //           (1 = Open valve, 0 = no action)
   // 
   //  CLOSE_CMD     Output to drive the valve to a closed state       Bool      Out
   //           (1 = Close valve, 0 = no action)
   //  ――――――――――――――――――――――――――――――――――――――――――
   // 
   //                ━━━   ⬙⬙⬙⬙⬙⬙   ━━━
   // 
   // 
   // 
   // ▄▄▄▄▄▄▄▄▄▄▄▄▄▄▄▄▄▄▄▄▄▄▄▄▄▄▄▄▄▄▄▄▄▄▄▄▄▄▄▄▄▄▄▄
   // 6.     DATA STRUCTURES AND USAGE
   // 
   // 
   // The block has the following associated data structure:
   // 
   // 
   //  ――――――――――――――――――――――――――――――――――――――――――
   //  DATA STRUCTURE             DESCRIPTION
   //  ――――――――――――――――――――――――――――――――――――――――――
   //  UT01000_St_SysRevision          Revision information for this block    See FC01101
   //  UT01101_St_SysLicence           Licence information for this block  See FC01101
   //  UT21000_Dy_SysSignals           System signals for logic and timing  See FC01101
   // 
   //  UT11101_St_DevValveBi        Static data that holds the configuration data
   //                     for the device (timer presets, limit switch 
   //                     and interlock configuration &c.)
   // 
   //  UT31101_Dy_DevValveBi          Dynamic data that holds the live data for the
   //                     device (its mode, status and messages and 
   //                     any other dynamic information required by the 
   //                     module)
   // 
   //  ――――――――――――――――――――――――――――――――――――――――――
   // 
   // 
   // 
   // ▂▂▂▂▂▂▂▂▂▂▂▂▂▂▂▂▂▂▂▂▂▂▂▂▂▂▂▂▂▂▂▂▂▂▂▂▂▂▂▂▂▂▂▂
   // 6.1     UT11101_St_DevValveBi
   // 
   // The static data structure for an isolating valve.
   // 
   // 
   //  UT11101_St_DevValveBi (full contents)
   //  ――――――――――――――――――――――――――――――――――――――――――
   //  SIGNAL NAME          FUNCTION                     TYPE
   //  ――――――――――――――――――――――――――――――――――――――――――
   //  CONFIG_MAINT_OP      CONFIG — Maintains or deenergises the outputs   Bool
   //                      (1 = maintain OP, 0 = deenergise OP)
   //  CONFIG_FBK_OPEN_EN    CONFIG — Open feedback is enabled        Bool
   //                      (1 = open feedback, 0 = no feedback)
   //  CONFIG_FBK_CLOSED_EN   CONFIG — Closed feedback is enabled         Bool
   //                      (1 = closed feedback, 0 = no feedback)
   //  CONFIG_ESTOP_DIS     CONFIG — E_STOP signal disabled           Bool
   //                      (1 = E_STOP not used, 0 = in use)
   //  CONFIG_TRIP_DIS      CONFIG — TRIP signal disabled           Bool
   //                      (1 = TRIP not used, 0 = in use)
   //  CONFIG_ILOCK_DIS     CONFIG — INTERLOCK signal disabled        Bool
   //                      (1 = INTERLOCK not used, 0 = in use)
   //  CONFIG_PERM_DIS      CONFIG — PERMISSIVE signal disabled         Bool
   //                      (1 = PERMISSIVE not used, 0 = in use)
   //  CONFIG_TRIP_OP_CL       CONFIG — TRIP state                  Bool
   //                      (1 = open, 0 = close)
   //  CONFIG_ILOCK_OP_CL      CONFIG — INTERLOCK state              Bool
   //                      (1 = open, 0 = close)
   //  CONFIG_PERM_OP_CL       CONFIG — PERMISSIVE permitted state         Bool
   //                      (1 = open, 0 = closed)
   //  CONFIG_FP_DIS               CONFIG — Faceplate is disabled           Bool
   //                      (1 = no Faceplate, 0 = normal)
   //  CONFIG_MAN_DIS              CONFIG — Manual mode is disabled          Bool
   //                      (1 = no manual mode, 0 = normal)
   //  CONFIG_BYPASS_DIS     CONFIG — Bypass mode is disabled           Bool
   //                      (1 = no bypass mode, 0 = normal)
   //  CONFIG_SIM_DIS             CONFIG — Simulation is disabled            Bool
   //                      (1 = no simulation, 0 = normal)
   //  CONFIG_RL_EN       CONFIG — Remote/local mode enabled       Bool
   //                      (1 = enabled, 0 = all mode)
   // 
   //  INFO_TAG          INFORMATION — Instrument ID tag          String[20]
   // 
   //  TIME_OPENING_MAX    TIMER — Initial value of opening operation timer      Real
   //                      (counts down from this value), [seconds]
   //  TIME_CLOSING_MAX       TIMER — Initial value of closing operation timer     Real
   //                      (counts down from this value), [seconds]
   //  TIME_OPENING_RUNON     TIMER — Initial value of opening run-on timer         Real
   //                      (counts down from this value), [seconds]
   //  TIME_CLOSING_RUNON        TIMER — Initial value of closing run-on timer           Real
   //                      (counts down from this value), [seconds]
   //  TIME_DER_OPEN              TIMER — Percentage of opening timer to expired      Real
   //                      before simulating FBK_OPEN, [percent]
   //  TIME_DER_CLOSED            TIMER — Percentage of closing timer to expired        Real
   //                      before simulating FBK_CLOSED, [percent]
   //  TIME_RECOVERY              TIMER — Initial value of the recovery timer      Real
   //                      (counts down from this value), [seconds]
   // 
   //  ――――――――――――――――――――――――――――――――――――――――――
   // 
   // 
   // 
   // ▂▂▂▂▂▂▂▂▂▂▂▂▂▂▂▂▂▂▂▂▂▂▂▂▂▂▂▂▂▂▂▂▂▂▂▂▂▂▂▂▂▂▂▂
   // 6.2      UT31101_Dy_DevValveBi
   // 
   // The static data structure for an isolating valve.
   // 
   // 
   // 
   //  UT31101_Dy_DevValveBi (full contents)
   //  ――――――――――――――――――――――――――――――――――――――――――
   //  SIGNAL NAME          FUNCTION                     TYPE
   //  ――――――――――――――――――――――――――――――――――――――――――
   //  status_Closed        STATUS — Valve is confirmed closed          Bool
   //                      (1 = closed, 0 = not closed)
   //  status_Open        STATUS — Valve is confirmed open         Bool
   //                      (1 = open, 0 = not open)
   //  status_Closing       STATUS — Valve is closing             Bool
   //                      (1 = closing, 0 = not closing)
   //  status_Opening        STATUS — Valve is opening              Bool
   //                      (1 = opening, 0 = not opening)
   //  status_Operating        STATUS — Valve is changing state           Bool
   //                      (1 = changing state, 0 = fixed state)
   //  status_Fault            STATUS — Valve is in fault              Bool
   //                      (1 = fault present, 0 = healthy)
   //  status_OpenOn        STATUS — Valve OPEN_CMD output is on        Bool
   //                      (1 = OPEN_CMD on, 0 = OPEN_CMD off)
   //  status_CloseOn        STATUS — Valve CLOSE_CMD output is on         Bool
   //                      (1 = CLOSE_CMD on, 0 = CLOSE_CMD off)
   //  status_Aut           STATUS — Automatic mode active           Bool
   //                      (1 = auto mode on, 0 = auto mode off)
   //  status_Man          STATUS — Manual mode active             Bool
   //                      (1 = man mode on, 0 = man mode off)
   //  status_EStop          STATUS — E_STOP safety signal is active         Bool
   //                      (1 = active, 0 = healthy)
   //  status_Trip        STATUS — TRIP signal is active             Bool
   //                      (1 = active, 0 = healthy)
   //  status_Ilock         STATUS — INTERLOCK signal is active            Bool
   //                      (1 = active, 0 = healthy)
   //  status_Perm        STATUS — PERMISSIVE signal is active           Bool
   //                      (1 = active, 0 = healthy)
   //  status_BypassOn        STATUS — Valve is in bypass mode          Bool
   //                      (1 = Simulation mode, 0 = normal)
   //  status_SimOn           STATUS — Valve is in simulation mode               Bool
   //                      (1 = Simulation mode, 0 = normal)
   //  status_RemoteOn       STATUS — Valve is in remote mode                  Bool
   //                      (1 = Remote mode, 0 = normal)
   //  status_LocalOn         STATUS — Valve is in local mode                    Bool
   //                      (1 = Local mode, 0 = normal)
   //  status_RLOff         STATUS — Valve is in ALL mode                   Bool
   //                      (1 = ALL mode, 0 = normal)
   // 
   //  msg_FailToOpen       MESSAGE — Alarm – “Fail to open” is active         Bool
   //  msg_FailToClose       MESSAGE — Alarm – “Fail to close” is active        Bool
   //  msg_FailWhileOpen    MESSAGE — Alarm – “Fail while open” is active      Bool
   //  msg_FailWhileClosed     MESSAGE — Alarm – “Fail while closed” is active   Bool
   //  msg_Flt_External         MESSAGE — Alarm – “external fault" is active      Bool
   // 
   //  mode_AutMan        MODE — Automatic or manual mode selection     Bool
   //                    (1 = auto mode active, 0 = man mode)
   //  mode_BypassOn      MODE — Bypass mode                Bool
   //                    (1 = bypass mode active, 0 = normal)
   //  mode_SimOn         MODE — Simulation mode               Bool
   //                    (1 = sim mode active, 0 = normal)
   //  mode_SimValue       MODE — Simulation value               Int
   //                    (0 = no limits, 1 = always open, 
   //                    2 = always closed, 3 = follow demand)
   //  mode_RemoteOn        MODE — Remote SCADA control enabled       Bool
   //                    (1 = active, 0 = disabled or N/A)
   //  mode_LocalOn         MODE — Local HMI control enabled           Bool
   //                    (1 = active, 0 = disabled or N/A)
   //  mode_Reset        MODE — Fault reset – 1 cycle only           Bool
   //                    (1 = Reset faults, 0 = does nothing)
   //  ctrl_Aut_OpenClose       CONTROL — Auto mode open or close valve     Bool
   //                          (1 = open valve , 0 = close valve)
   //  ctrl_Man_OpenClose      CONTROL — Manual mode open or close valve   Bool
   //                          (1 = open valve , 0 = close valve)
   // 
   //  batch_ID         BATCH — Booking ID (optional for batch operations)   UInt
   // 
   //  actual_Operating_Timer     ACTUAL — Timer value — operating opening/closing  Real
   //                      timer actual value [seconds]
   //  actual_Runon_Timer      ACTUAL — Timer value — run-on opening/closing  Real
   //                      timer actual value [seconds]
   //  actual_Recovery_Timer     ACTUAL — Timer value — recovery timer         Real
   //                      timer actual value [seconds]
   //  actual_Last_Op_Time       ACTUAL — actual time taken to achieve the last    Real
   //                      good valve position [seconds]
   // 
   //  $derived_fbk_open     INTERNAL — Derived feedback open signal       Bool
   //                          (1 = open , 0 = not open)
   //  $derived_fbk_closed      INTERNAL — Derived feedback closed signal        Bool
   //                          (1 = closed, 0 = not closed)
   //  $sim_fbk_open         INTERNAL — Simulated feedback open signal         Bool
   //                          (1 = open , 0 = not open)
   //  $sim_fbk_closed          INTERNAL — Simulated feedback closed signal      Bool
   //                          (1 = closed, 0 = not closed)
   //  $ctrl_OpenClose       INTERNAL — actual open or close request,         Bool
   //                          incorporates all priorities
   //                         (1 = open valve, 0 = close valve)
   //  $pret_Open             INTERNAL — Edge retention (+ve) rising edge of    Bool
   //                          ctrl_OpenClose (change to opening)
   //  $nret_Close            INTERNAL — Edge retention (-ve) falling edge of        Bool
   //                          ctrl_OpenClose (change to closing)
   //  ――――――――――――――――――――――――――――――――――――――――――
   // 
   // 
   // With the exception of the flowing, all these signals are discussed in the previous sections, the 
   // outstanding items are firstly:
   // 
   //      batch_ID
   // 
   // The batch_ID is not required for normal use; it is only used where a “booking” system is used 
   // (common in batch and routing applications). Such booking applications can acquire the device 
   // if it is free and reserve it for a particular phase of the batch. Batch applications are a topic in 
   // their own right and are discussed separately in the online User Guide.
   // 
   // There are internal working signals (all signals the start with a $ are internal working signals used 
   // by the module). In this instance they are used as follows: 
   //  
   // The $derived_fbk_open and $derived_fbk_closed are the internally derived open and closed 
   // feedback signal used in place of FBK_OPEN and FBK_CLOSED if either CONFIG_FBK_OPEN_EN 
   // or CONFIG_FBK_CLOSED_EN is set to zero.
   // 
   // The $sim_fbk_open and $sim_fbk_closed are the simulated position feedback signal used in 
   // place of FBK_OPEN and FBK_CLOSED if simulation mode is active.
   // 
   // $ctrl_OpenClose is the required state of the valve, it takes into account the auto/manual 
   // requested state and modifies this according to any interlocks, safety signals or faults that 
   // may be present.
   // 
   // The $pret_Open and $nret_Close are edge retention signals used to detect either a rising 
   // (a change to opening) or a falling (a change to closing) edge on the $ctrl_OpenClose signal.
   // 
   // 
   //                ━━━   ⬙⬙⬙⬙⬙⬙   ━━━
   // 
   // 
   // 
   // ▄▄▄▄▄▄▄▄▄▄▄▄▄▄▄▄▄▄▄▄▄▄▄▄▄▄▄▄▄▄▄▄▄▄▄▄▄▄▄▄▄▄▄▄
   // 7.     CONSTANTS AND TEMPORARY (LOCAL) DATA
   // 
   // 
   // 
   // ▂▂▂▂▂▂▂▂▂▂▂▂▂▂▂▂▂▂▂▂▂▂▂▂▂▂▂▂▂▂▂▂▂▂▂▂▂▂▂▂▂▂▂▂
   // 7.1     Constants
   // 
   // 
   // The following constants data is used:
   // 
   //  ――――――――――――――――――――――――――――――――――――――――――
   //  SIGNAL NAME       Value    FUNCTION                  TYPE
   //  ――――――――――――――――――――――――――――――――――――――――――
   //  k_TIME_OP_MIN      0.21      Minimum value for the operation timer     Real
   //  k_TIME_SIM_MIN     0.21      Elapsed op timer value for sim mode 3        Real
   //  ――――――――――――――――――――――――――――――――――――――――――
   // 
   // 
   // 
   // ▂▂▂▂▂▂▂▂▂▂▂▂▂▂▂▂▂▂▂▂▂▂▂▂▂▂▂▂▂▂▂▂▂▂▂▂▂▂▂▂▂▂▂▂
   // 7.2     Temporary (local) data
   // 
   // 
   // The following temporary data is used:
   // 
   //  ――――――――――――――――――――――――――――――――――――――――――
   //  SIGNAL NAME          FUNCTION                  TYPE
   //  ――――――――――――――――――――――――――――――――――――――――――
   //  revInfo             Revision information for the block         UT01000
   //  licInfo           Licensing information for the block      UT01101
   //  calClosedElapsedTime     Calc - Derived closed signal elapsed time   Real
   //  calOpenElapsedTime       Calc - Derived open signal elapsed time   Real
   //  wrkOpen            Working - open position feedback signal      Bool
   //  wrkClosed         Working - closed position feedback signal   Bool
   //  wrkCtrlPriority40        Working - priority 40 controls the valve      Bool
   //  wrkCtrlPriority30        Working - priority 30 controls the valve      Bool
   //  wrkCtrlPriority20        Working - priority 20 controls the valve      Bool
   //  wrkCtrlPriority10        Working - priority 10 controls the valve      Bool
   //  wrkCtrlPriority00        Working - priority 00 controls the valve      Bool
   //  wrkCtrlAutManOpCl     Working - aut/man open or close request     Bool
   //  wrkTimeFbkOpenSim     Working - Err checked TIME_FBK_OPEN            Real
   //  wrkTimeFbkClosedSim     Working - Err checked TIME_FBK_CLOSED           Real
   //  wrkInt           Working storage area (integer)          Int
   //  wrkReal           Working storage (Real)             Real
   //  wrkDInt           Working storage area (double integer)         DInt
   //  ――――――――――――――――――――――――――――――――――――――――――
   // 
   //                ━━━   ⬙⬙⬙⬙⬙⬙   ━━━
   // 
   // 
   // 
   // ▄▄▄▄▄▄▄▄▄▄▄▄▄▄▄▄▄▄▄▄▄▄▄▄▄▄▄▄▄▄▄▄▄▄▄▄▄▄▄▄▄▄▄▄
   // 8.     BLOCK CALLS AND ASSOCIATIONS
   // 
   // 
   // This section details any blocks which may be called from within this software module (subroutine 
   // functions for example), any partner blocks with which it may be associated (for example a 
   // receive module that is partner with a transmit module &c.). It lists any system functions which 
   // may be called (e.g. reading the real time clock) and any system data types that may be used.
   // 
   // Finally, it lists any special calling requirements for the block (for example, must be called from 
   // within a cyclic interrupt organisation block) and if the block is using “optimised access” (this is 
   // the default arrangement).
   // 
   // 
   // 
   // ▂▂▂▂▂▂▂▂▂▂▂▂▂▂▂▂▂▂▂▂▂▂▂▂▂▂▂▂▂▂▂▂▂▂▂▂▂▂▂▂▂▂▂▂
   // 8.1     Block calls from within this module
   // 
   // 
   // There are no PAL block calls from within this block.
   // 
   // 
   // 
   // ▂▂▂▂▂▂▂▂▂▂▂▂▂▂▂▂▂▂▂▂▂▂▂▂▂▂▂▂▂▂▂▂▂▂▂▂▂▂▂▂▂▂▂▂
   // 8.2     Blocks associated with this module
   // 
   // 
   // This is a stand-alone block and is not associated with any other blocks.
   // 
   // 
   // 
   // ▂▂▂▂▂▂▂▂▂▂▂▂▂▂▂▂▂▂▂▂▂▂▂▂▂▂▂▂▂▂▂▂▂▂▂▂▂▂▂▂▂▂▂▂
   // 8.3     System block calls and system data types
   // 
   // There are no system block calls
   // 
   // 
   // 
   // ▂▂▂▂▂▂▂▂▂▂▂▂▂▂▂▂▂▂▂▂▂▂▂▂▂▂▂▂▂▂▂▂▂▂▂▂▂▂▂▂▂▂▂▂
   // 8.4     Special properties and requirements
   // 
   // 
   // 
   // ▁▁▁▁▁▁▁▁▁▁▁▁▁▁▁▁▁▁▁▁▁▁▁▁▁▁▁▁▁▁▁▁▁▁▁▁▁▁▁▁▁▁▁▁
   // 8.4.1     Block optimisation, IEC compatibility and library conformance
   // 
   // 
   //    •   Block optimisation is ACTIVE for this block.
   // 
   //    •   The block has been checked for IEC compatibility and is compliant.
   // 
   //    •   The block is compatible with all IEC library-conformance module constraints
   // 
   // 
   // 
   // ▁▁▁▁▁▁▁▁▁▁▁▁▁▁▁▁▁▁▁▁▁▁▁▁▁▁▁▁▁▁▁▁▁▁▁▁▁▁▁▁▁▁▁▁
   // 8.4.2     Calling requirements
   // 
   // 
   // There are no special calling requirements for this block.
   // 
   //                ━━━   ⬙⬙⬙⬙⬙⬙   ━━━
   // 
   // 
   // 
   // ▄▄▄▄▄▄▄▄▄▄▄▄▄▄▄▄▄▄▄▄▄▄▄▄▄▄▄▄▄▄▄▄▄▄▄▄▄▄▄▄▄▄▄▄
   // 9.     EXAMPLE USAGE
   // 
   // 
   // The following shows a typical deployment of FC11101:
   // 
   //                         ┌─────────────
   //      ───────────────────┤ FC11101 
   //                         ├───────────────┤
   //    "DB21101_DY_StdGlobalData".SysSignals ─┤ SYS_SIGNALS            %Q1.0
   //                         │            OPEN_CMD ├─  "V001_OPEN_CMD"
   //                   %I1.2     │               │
   //                 "V001_FBK_OPEN" ─┤ FBK_OPEN             │  %Q1.1
   //                         │          CLOSE_CMD ├─  "V001_CLOSE_CMD"
   //                   %I1.1     │               │
   //               "V001_FBK_CLOSED" ─┤ FBK_CLOSED            │
   //                         │               │
   //            %I1.0            │               │
   //           "V001_FAULT"             │               │
   //        ────┤╱├──────────┤ EXT_FAULT                │
   //                         │               │
   //            %I1.4            │               │
   //          "ZONEA_ESTOP"               │               │
   //        ────┤╱├──────────┤ E_STOP                │
   //                         │               │
   //                    "_False" ─┤ TRIP                    │
   //                         │               │
   //            "DB23002_Dy_ILock.V001"─┤ INTERLOCK             │
   //                         │               │
   //                    "_False" ─┤ PERMISSIVE            │
   //                         │               │
   //                         │               │
   //                         │               │
   //            "DB11101_St_DevValveBi".V001 ─┤ STATIC_DATA             │
   //                         │
   //            "DB31101_Dy_DevValveBi".V001 ─┤ DYNAMIC_DATA
   //                         │
   //                         │
   //                                         │
   //                                ─────────┘
   // 
   // 
   //               ━━━   ⬙⬙⬙⬙⬙⬙   ━━━
   // 
   // 
   // 
   // ▄▄▄▄▄▄▄▄▄▄▄▄▄▄▄▄▄▄▄▄▄▄▄▄▄▄▄▄▄▄▄▄▄▄▄▄▄▄▄▄▄▄▄▄
   // 10.     TEST AND VERIFICATION PATH
   // 
   // 
   // The following diagram shows the full test and verification path for the formal release of each 
   // version of the software module. See the Test Plan [Ref. 003] for full details, available here:
   //         https://psop.uk/pal-tp-p
   // 
   // 
   //         FC11101-T001
   // 
   //     Test version: 000.801
   //  Released version: 001.000
   // Released commit: D0016 
   // 
   //        SCR      SMT 
   // ＿＿＿＿＿＿┌┐＿＿ ▛▜ ＿
   //       └┘   ▙▟  
   // Initial test           
   // 
   // Initial test to release the      Comments updated & 
   // module following the      minor typographical 
   // development stage.       corrections
   // Full SMT              SCV only
   // 
   // 
   // Where:
   // ――――――――――――――――――――――――――――――――――――――――――――
   //  SCR    Source Code Review      A visual inspection of the software to ensure it has been written  
   // ┌┐             to the correct standards, uses the correct structures within the
   // └┘             software and is generally suitable for deployment.               
   // 
   //  SMT Software Module Test    A full and detailed test of an individual software module in
   //   ▛▜              isolation; such testing requires that all branches of the 
   //   ▙▟              software are tested. 
   // 
   //                It tests all the interfaces to the module, any data recorded or 
   //                stored by the module, all error and exception handling functions 
   //                and tests all timed and interrupt driven operations.
   // 
   //  SCV Software Compatibility     A mechanism for verifying that no executable code software 
   // ╓╖    Verification          changes have been made to a module following changes to
   // ╙╜             comment fields.
   // 
   //                Allows typographical errors &c. to be corrected without forcing 
   //                a full SMT on a module that has not functionally changed.
   // ――――――――――――――――――――――――――――――――――――――――――――
   // 
   // An SCV can only be performed on a module that has at some point previously, successfully 
   // completed both an SCR and SMT. Where an SCV is implemented, it replaces the requirement for 
   // both the SCR and the SMT for the test iteration in question.
   // 
   //                ━━━   ⬙⬙⬙⬙⬙⬙   ━━━
   // 
   // 
   // ██████████████ █ █ █ █  END   █ █ █ █ ██████████████
END_REGION

REGION Network 7: Current revision and modification history
   // ▄▄▄▄▄▄▄▄▄▄▄▄▄▄▄▄▄▄▄▄▄▄▄▄▄▄▄▄▄▄▄▄▄▄▄▄▄▄▄▄▄▄▄▄
   // MODIFICATION HISTORY
   // 
   // 
   // The revision data shown here, in the network comments, contains additional information 
   // reflecting the software development workflow under the version control system (VCS) employed 
   // to track all software changes.
   // 
   // The VCS in use is the Git Source Code Management system in conjunction with the GitHub online 
   // hosting system. The software in its entirety is available in the GitHub remote repository:
   // 
   //      https://github.com/practicalseries/PS2001-pal-software
   // 
   // The repository is public and can be freely copied (forked in GitHub terminology) and used 
   // under the MIT licence. 
   // 
   // The MIT licence is reproduced in full in the last network of this software module.
   // 
   // 
   //  ―――――――――――――――――――――――――――――――――――――――――――
   //  DATE       REVISION             MASTER BRANCH     DEV
   //          (nnn.amm)   COMMIT TAG    (Base ---> Merge)    BRANCH   Author
   //  ———————————————————————————————————————————
   //  2023.02.01    000.801   D0015A-000.801   D0015 N/A     D0015A   M. Gledhill
   //                        FC11101  — Released for test (SMTS)
   // 
   //  2023.01.28    000.102   D0015A-000.102   D0015 N/A     D0015A   M. Gledhill
   //                        FC11101  — Incremental build
   // 
   //  2022.08.15    000.101   D0015A-000.101   D0015 N/A     D0015A   M. Gledhill
   //                        FC11101 — Block created, Comments added
   //  ———————————————————————————————————————————
   //   Where: nnn  =  Major revision
   //         a  =  Type (1-7 Development, 8 Proving, 9 Qualification, 0 Release)
   //       mm  =  Minor revision (must be 00 if a = 0)
   //         Block properties version number should be set to nn.a (only one decimal place)
   // 
   // ▄▄▄▄▄▄▄▄▄▄▄▄▄▄▄▄▄▄▄▄▄▄▄▄▄▄▄▄▄▄▄▄▄▄▄▄▄▄▄▄▄▄▄▄
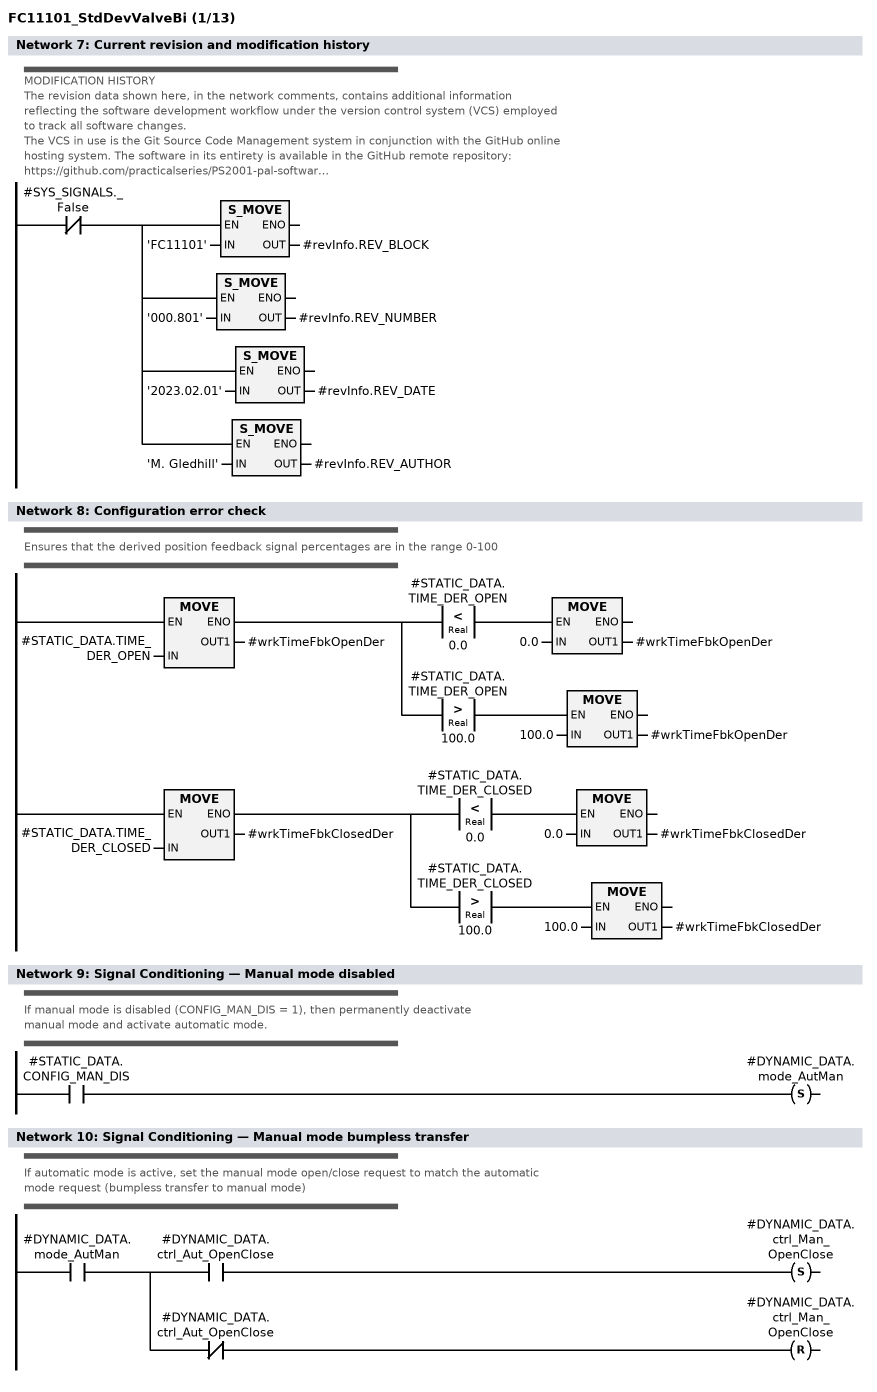
   RUNG wire#powerrail
      I_Contact( #SYS_SIGNALS._False )
      wire#w1
      S_Move(in := 'FC11101', out => #revInfo.REV_BLOCK)
   END_RUNG
   RUNG wire#w1
      S_Move(in := '000.801', out => #revInfo.REV_NUMBER)
   END_RUNG
   RUNG wire#w1
      S_Move(in := '2023.02.01', out => #revInfo.REV_DATE)
   END_RUNG
   RUNG wire#w1
      S_Move(in := 'M. Gledhill', out => #revInfo.REV_AUTHOR)
   END_RUNG
   // the same network as SCL:
   IF NOT #SYS_SIGNALS._False THEN
       #revInfo.REV_BLOCK := 'FC11101';
       #revInfo.REV_NUMBER := '000.801';
       #revInfo.REV_DATE := '2023.02.01';
       #revInfo.REV_AUTHOR := 'M. Gledhill';
   END_IF;
END_REGION

REGION Network 8: Configuration error check
   // ▀▀▀▀▀▀▀▀▀▀▀▀▀▀▀▀▀▀▀▀▀▀▀▀▀▀▀▀▀▀▀▀▀▀▀▀▀▀▀▀▀▀▀▀
   // Ensures that the derived position feedback signal percentages are in the range 0-100
   // ▄▄▄▄▄▄▄▄▄▄▄▄▄▄▄▄▄▄▄▄▄▄▄▄▄▄▄▄▄▄▄▄▄▄▄▄▄▄▄▄▄▄▄▄
   RUNG wire#powerrail
      Move(in := #STATIC_DATA.TIME_DER_OPEN, out1 => #wrkTimeFbkOpenDer)
      wire#w1
      { S7_Templates := "SrcType := Real" } LT_Contact(in1 := #STATIC_DATA.TIME_DER_OPEN, in2 := 0.0)
      Move(in := 0.0, out1 => #wrkTimeFbkOpenDer)
   END_RUNG
   RUNG wire#w1
      { S7_Templates := "SrcType := Real" } GT_Contact(in1 := #STATIC_DATA.TIME_DER_OPEN, in2 := 100.0)
      Move(in := 100.0, out1 => #wrkTimeFbkOpenDer)
   END_RUNG
   RUNG wire#powerrail
      Move(in := #STATIC_DATA.TIME_DER_CLOSED, out1 => #wrkTimeFbkClosedDer)
      wire#w2
      { S7_Templates := "SrcType := Real" } LT_Contact(in1 := #STATIC_DATA.TIME_DER_CLOSED, in2 := 0.0)
      Move(in := 0.0, out1 => #wrkTimeFbkClosedDer)
   END_RUNG
   RUNG wire#w2
      { S7_Templates := "SrcType := Real" } GT_Contact(in1 := #STATIC_DATA.TIME_DER_CLOSED, in2 := 100.0)
      Move(in := 100.0, out1 => #wrkTimeFbkClosedDer)
   END_RUNG
   // the same network as SCL:
   #wrkTimeFbkOpenDer := #STATIC_DATA.TIME_DER_OPEN;
   IF #STATIC_DATA.TIME_DER_OPEN < 0.0 THEN #wrkTimeFbkOpenDer := 0.0; END_IF;
   IF #STATIC_DATA.TIME_DER_OPEN > 100.0 THEN #wrkTimeFbkOpenDer := 100.0; END_IF;
   #wrkTimeFbkClosedDer := #STATIC_DATA.TIME_DER_CLOSED;
   IF #STATIC_DATA.TIME_DER_CLOSED < 0.0 THEN #wrkTimeFbkClosedDer := 0.0; END_IF;
   IF #STATIC_DATA.TIME_DER_CLOSED > 100.0 THEN #wrkTimeFbkClosedDer := 100.0; END_IF;
END_REGION

REGION Network 9: Signal Conditioning — Manual mode disabled
   // ▀▀▀▀▀▀▀▀▀▀▀▀▀▀▀▀▀▀▀▀▀▀▀▀▀▀▀▀▀▀▀▀▀▀▀▀▀▀▀▀▀▀▀▀
   // If manual mode is disabled (CONFIG_MAN_DIS = 1), then permanently deactivate
   // manual mode and activate automatic mode.
   // ▄▄▄▄▄▄▄▄▄▄▄▄▄▄▄▄▄▄▄▄▄▄▄▄▄▄▄▄▄▄▄▄▄▄▄▄▄▄▄▄▄▄▄▄
   RUNG wire#powerrail
      Contact( #STATIC_DATA.CONFIG_MAN_DIS )
      S_Coil( #DYNAMIC_DATA.mode_AutMan )
   END_RUNG
   // the same network as SCL:
   IF #STATIC_DATA.CONFIG_MAN_DIS THEN #DYNAMIC_DATA.mode_AutMan := TRUE; END_IF;
END_REGION

REGION Network 10: Signal Conditioning — Manual mode bumpless transfer
   // ▀▀▀▀▀▀▀▀▀▀▀▀▀▀▀▀▀▀▀▀▀▀▀▀▀▀▀▀▀▀▀▀▀▀▀▀▀▀▀▀▀▀▀▀
   // If automatic mode is active, set the manual mode open/close request to match the automatic
   // mode request (bumpless transfer to manual mode)
   // ▄▄▄▄▄▄▄▄▄▄▄▄▄▄▄▄▄▄▄▄▄▄▄▄▄▄▄▄▄▄▄▄▄▄▄▄▄▄▄▄▄▄▄▄
   RUNG wire#powerrail
      Contact( #DYNAMIC_DATA.mode_AutMan )
      wire#w1
      Contact( #DYNAMIC_DATA.ctrl_Aut_OpenClose )
      S_Coil( #DYNAMIC_DATA.ctrl_Man_OpenClose )
   END_RUNG
   RUNG wire#w1
      I_Contact( #DYNAMIC_DATA.ctrl_Aut_OpenClose )
      R_Coil( #DYNAMIC_DATA.ctrl_Man_OpenClose )
   END_RUNG
   // the same network as SCL:
   IF #DYNAMIC_DATA.mode_AutMan AND #DYNAMIC_DATA.ctrl_Aut_OpenClose THEN
       #DYNAMIC_DATA.ctrl_Man_OpenClose := TRUE;
   END_IF;
   IF #DYNAMIC_DATA.mode_AutMan AND NOT #DYNAMIC_DATA.ctrl_Aut_OpenClose THEN
       #DYNAMIC_DATA.ctrl_Man_OpenClose := FALSE;
   END_IF;
END_REGION

REGION Network 11: Signal Conditioning — Bypass mode disabled
   // ▀▀▀▀▀▀▀▀▀▀▀▀▀▀▀▀▀▀▀▀▀▀▀▀▀▀▀▀▀▀▀▀▀▀▀▀▀▀▀▀▀▀▀▀
   // If bypass mode is disabled (CONFIG_BYPASS_DIS = 1), then permanently deactivate
   // bypass mode.
   // ▄▄▄▄▄▄▄▄▄▄▄▄▄▄▄▄▄▄▄▄▄▄▄▄▄▄▄▄▄▄▄▄▄▄▄▄▄▄▄▄▄▄▄▄
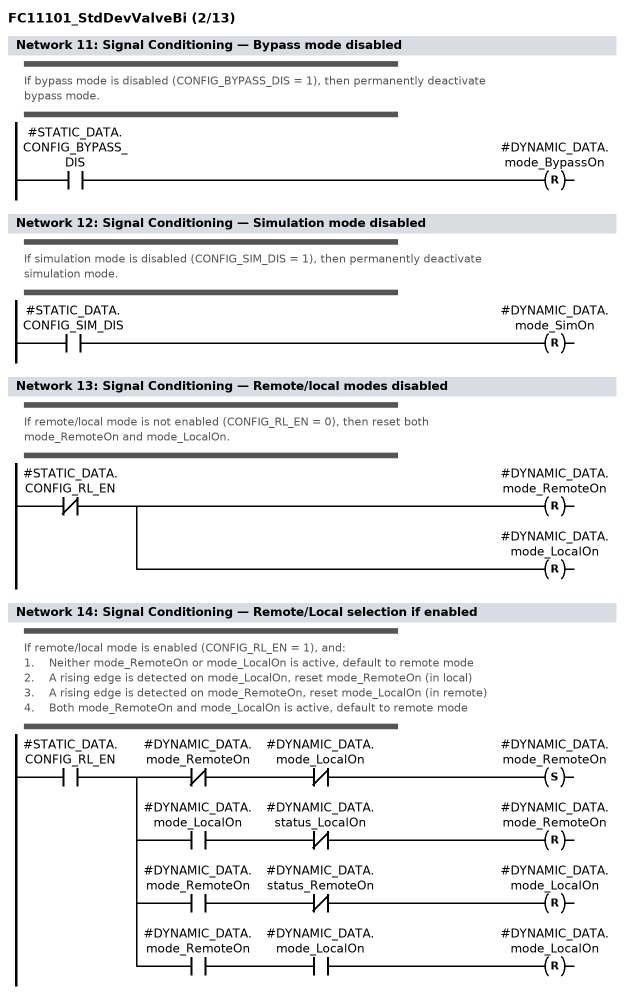
   RUNG wire#powerrail
      Contact( #STATIC_DATA.CONFIG_BYPASS_DIS )
      R_Coil( #DYNAMIC_DATA.mode_BypassOn )
   END_RUNG
   // the same network as SCL:
   IF #STATIC_DATA.CONFIG_BYPASS_DIS THEN #DYNAMIC_DATA.mode_BypassOn := FALSE; END_IF;
END_REGION

REGION Network 12: Signal Conditioning — Simulation mode disabled
   // ▀▀▀▀▀▀▀▀▀▀▀▀▀▀▀▀▀▀▀▀▀▀▀▀▀▀▀▀▀▀▀▀▀▀▀▀▀▀▀▀▀▀▀▀
   // If simulation mode is disabled (CONFIG_SIM_DIS = 1), then permanently deactivate
   // simulation mode.
   // ▄▄▄▄▄▄▄▄▄▄▄▄▄▄▄▄▄▄▄▄▄▄▄▄▄▄▄▄▄▄▄▄▄▄▄▄▄▄▄▄▄▄▄▄
   RUNG wire#powerrail
      Contact( #STATIC_DATA.CONFIG_SIM_DIS )
      R_Coil( #DYNAMIC_DATA.mode_SimOn )
   END_RUNG
   // the same network as SCL:
   IF #STATIC_DATA.CONFIG_SIM_DIS THEN #DYNAMIC_DATA.mode_SimOn := FALSE; END_IF;
END_REGION

REGION Network 13: Signal Conditioning — Remote/local modes disabled
   // ▀▀▀▀▀▀▀▀▀▀▀▀▀▀▀▀▀▀▀▀▀▀▀▀▀▀▀▀▀▀▀▀▀▀▀▀▀▀▀▀▀▀▀▀
   // If remote/local mode is not enabled (CONFIG_RL_EN = 0), then reset both 
   // mode_RemoteOn and mode_LocalOn.
   // ▄▄▄▄▄▄▄▄▄▄▄▄▄▄▄▄▄▄▄▄▄▄▄▄▄▄▄▄▄▄▄▄▄▄▄▄▄▄▄▄▄▄▄▄
   RUNG wire#powerrail
      I_Contact( #STATIC_DATA.CONFIG_RL_EN )
      wire#w1
      R_Coil( #DYNAMIC_DATA.mode_RemoteOn )
   END_RUNG
   RUNG wire#w1
      R_Coil( #DYNAMIC_DATA.mode_LocalOn )
   END_RUNG
   // the same network as SCL:
   IF NOT #STATIC_DATA.CONFIG_RL_EN THEN
       #DYNAMIC_DATA.mode_RemoteOn := FALSE;
       #DYNAMIC_DATA.mode_LocalOn := FALSE;
   END_IF;
END_REGION

REGION Network 14: Signal Conditioning — Remote/Local selection if enabled
   // ▀▀▀▀▀▀▀▀▀▀▀▀▀▀▀▀▀▀▀▀▀▀▀▀▀▀▀▀▀▀▀▀▀▀▀▀▀▀▀▀▀▀▀▀
   // If remote/local mode is enabled (CONFIG_RL_EN = 1), and:
   // 
   //    1.  Neither mode_RemoteOn or mode_LocalOn is active, default to remote mode
   //    2.  A rising edge is detected on mode_LocalOn, reset mode_RemoteOn (in local)
   //    3.  A rising edge is detected on mode_RemoteOn, reset mode_LocalOn (in remote)
   //    4.  Both mode_RemoteOn and mode_LocalOn is active, default to remote mode
   // ▄▄▄▄▄▄▄▄▄▄▄▄▄▄▄▄▄▄▄▄▄▄▄▄▄▄▄▄▄▄▄▄▄▄▄▄▄▄▄▄▄▄▄▄
   RUNG wire#powerrail
      Contact( #STATIC_DATA.CONFIG_RL_EN )
      wire#w1
      I_Contact( #DYNAMIC_DATA.mode_RemoteOn )
      I_Contact( #DYNAMIC_DATA.mode_LocalOn )
      S_Coil( #DYNAMIC_DATA.mode_RemoteOn )
   END_RUNG
   RUNG wire#w1
      Contact( #DYNAMIC_DATA.mode_LocalOn )
      I_Contact( #DYNAMIC_DATA.status_LocalOn )
      R_Coil( #DYNAMIC_DATA.mode_RemoteOn )
   END_RUNG
   RUNG wire#w1
      Contact( #DYNAMIC_DATA.mode_RemoteOn )
      I_Contact( #DYNAMIC_DATA.status_RemoteOn )
      R_Coil( #DYNAMIC_DATA.mode_LocalOn )
   END_RUNG
   RUNG wire#w1
      Contact( #DYNAMIC_DATA.mode_RemoteOn )
      Contact( #DYNAMIC_DATA.mode_LocalOn )
      R_Coil( #DYNAMIC_DATA.mode_LocalOn )
   END_RUNG
   // the same network as SCL:
   IF #STATIC_DATA.CONFIG_RL_EN AND NOT #DYNAMIC_DATA.mode_RemoteOn AND NOT #DYNAMIC_DATA.mode_LocalOn THEN
       #DYNAMIC_DATA.mode_RemoteOn := TRUE;
   END_IF;
   IF #STATIC_DATA.CONFIG_RL_EN AND #DYNAMIC_DATA.mode_LocalOn AND NOT #DYNAMIC_DATA.status_LocalOn THEN
       #DYNAMIC_DATA.mode_RemoteOn := FALSE;
   END_IF;
   IF #STATIC_DATA.CONFIG_RL_EN AND #DYNAMIC_DATA.mode_RemoteOn AND NOT #DYNAMIC_DATA.status_RemoteOn THEN
       #DYNAMIC_DATA.mode_LocalOn := FALSE;
   END_IF;
   IF #STATIC_DATA.CONFIG_RL_EN AND #DYNAMIC_DATA.mode_RemoteOn AND #DYNAMIC_DATA.mode_LocalOn THEN
       #DYNAMIC_DATA.mode_LocalOn := FALSE;
   END_IF;
END_REGION

REGION Network 15: Signal Conditioning — Derived open position
   // ▀▀▀▀▀▀▀▀▀▀▀▀▀▀▀▀▀▀▀▀▀▀▀▀▀▀▀▀▀▀▀▀▀▀▀▀▀▀▀▀▀▀▀▀
   // If there is no open position feedback (CONFIG_FBK_OPEN_EN = 0), then the open state of the 
   // valve is derived from the elapsed time of the operation timer using the following formulae:
   // 
   // ┌───────────────────────────────────────────┐
   // │$derived_fbk_open =1 when:                                │
   // │                                 wrkTimeFbkOpenDer  │
   // │actual_Operating_Timer ≤ TIME_OPENING_MAX ─ TIME_OPENING_MAX ╳ ----------------------------------------│
   // │                                     100     │
   // └───────────────────────────────────────────┘
   // Note:    wrkTimeFbkOpenDer is the error checked equivalent of TIME_FBK_OPEN
   // 
   // If the calculated elapsed time is close to or less than k_TIME_OP_MIN (210ms),
   // the calculated elapsed time (calOpenElapsedTime) is set to k_TIME_OP_MIN. This ensures at
   // least one timing pulse is required before the timer reaches zero.
   // 
   // The derived open signal ($derived_fbk_open) is reset if the valve is requested to be closed
   // ($ctrl_OpenClose = 0).
   // ▄▄▄▄▄▄▄▄▄▄▄▄▄▄▄▄▄▄▄▄▄▄▄▄▄▄▄▄▄▄▄▄▄▄▄▄▄▄▄▄▄▄▄▄
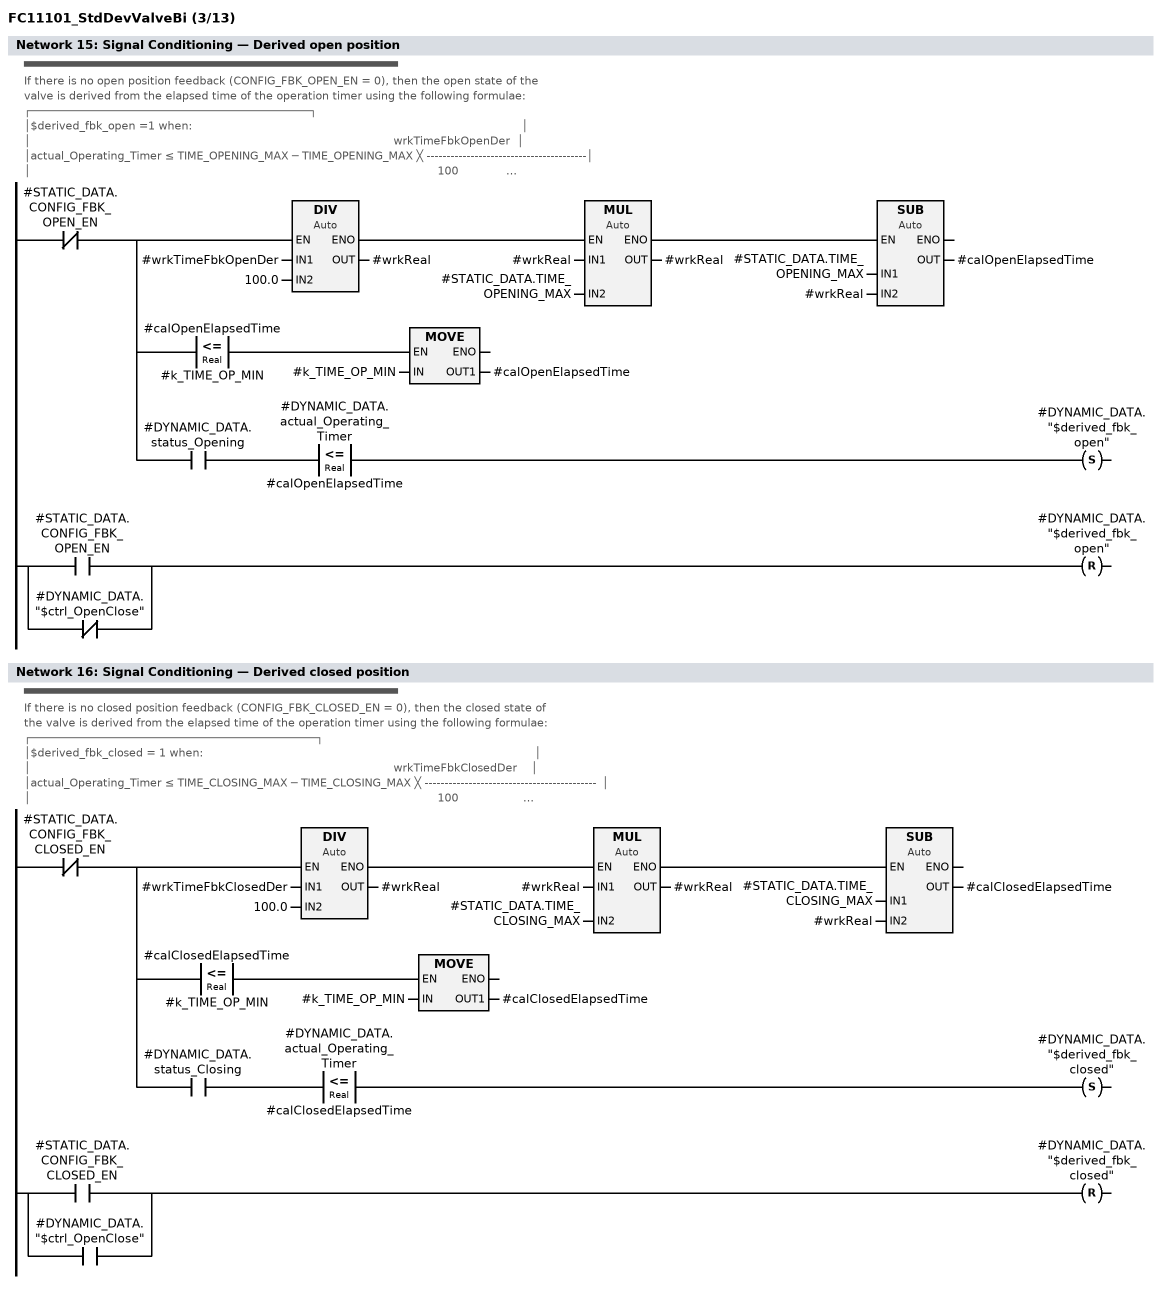
   RUNG wire#powerrail
      I_Contact( #STATIC_DATA.CONFIG_FBK_OPEN_EN )
      wire#w1
      Div(in1 := #wrkTimeFbkOpenDer, in2 := 100.0, out => #wrkReal)
      Mul(in1 := #wrkReal, in2 := #STATIC_DATA.TIME_OPENING_MAX, out => #wrkReal)
      Sub(in1 := #STATIC_DATA.TIME_OPENING_MAX, in2 := #wrkReal, out => #calOpenElapsedTime)
   END_RUNG
   RUNG wire#w1
      { S7_Templates := "SrcType := Real" } LE_Contact(in1 := #calOpenElapsedTime, in2 := #k_TIME_OP_MIN)
      Move(in := #k_TIME_OP_MIN, out1 => #calOpenElapsedTime)
   END_RUNG
   RUNG wire#w1
      Contact( #DYNAMIC_DATA.status_Opening )
      { S7_Templates := "SrcType := Real" } LE_Contact(in1 := #DYNAMIC_DATA.actual_Operating_Timer, in2 := #calOpenElapsedTime)
      S_Coil( #DYNAMIC_DATA."$derived_fbk_open" )
   END_RUNG
   RUNG wire#powerrail
      Contact( #STATIC_DATA.CONFIG_FBK_OPEN_EN )
      wire#w2
      R_Coil( #DYNAMIC_DATA."$derived_fbk_open" )
   END_RUNG
   RUNG wire#powerrail
      I_Contact( #DYNAMIC_DATA."$ctrl_OpenClose" )
   END_RUNG wire#w2
   // the same network as SCL:
   #_w1 := NOT #STATIC_DATA.CONFIG_FBK_OPEN_EN;
   IF #_w1 THEN
       #wrkReal := #wrkTimeFbkOpenDer / 100.0;
       #wrkReal := #wrkReal * #STATIC_DATA.TIME_OPENING_MAX;
       #calOpenElapsedTime := #STATIC_DATA.TIME_OPENING_MAX - #wrkReal;
   END_IF;
   IF #_w1 AND (#calOpenElapsedTime <= #k_TIME_OP_MIN) THEN #calOpenElapsedTime := #k_TIME_OP_MIN; END_IF;
   IF #_w1 AND #DYNAMIC_DATA.status_Opening AND (#DYNAMIC_DATA.actual_Operating_Timer <= #calOpenElapsedTime) THEN
       #DYNAMIC_DATA."$derived_fbk_open" := TRUE;
   END_IF;
   IF #STATIC_DATA.CONFIG_FBK_OPEN_EN OR NOT #DYNAMIC_DATA."$ctrl_OpenClose" THEN
       #DYNAMIC_DATA."$derived_fbk_open" := FALSE;
   END_IF;
END_REGION

REGION Network 16: Signal Conditioning — Derived closed position
   // ▀▀▀▀▀▀▀▀▀▀▀▀▀▀▀▀▀▀▀▀▀▀▀▀▀▀▀▀▀▀▀▀▀▀▀▀▀▀▀▀▀▀▀▀
   // If there is no closed position feedback (CONFIG_FBK_CLOSED_EN = 0), then the closed state of 
   // the valve is derived from the elapsed time of the operation timer using the following formulae:
   // 
   // ┌────────────────────────────────────────────┐
   // │$derived_fbk_closed = 1 when:                                 │
   // │                                 wrkTimeFbkClosedDer    │
   // │actual_Operating_Timer ≤ TIME_CLOSING_MAX ─ TIME_CLOSING_MAX ╳ -------------------------------------------  │
   // │                                     100            │
   // └────────────────────────────────────────────┘
   // Note:    wrkTimeFbkClosedDer is the error checked equivalent of TIME_FBK_CLOSED
   // 
   // If the calculated elapsed time is close to or less than k_TIME_OP_MIN (210ms),
   // the calculated elapsed time (calClosedElapsedTime) is set to k_TIME_OP_MIN. This ensures at
   // least one timing pulse is required before the timer reaches zero.
   // 
   // The derived closed signal ($derived_fbk_closed) is reset if the valve is requested to be open
   // ($ctrl_OpenClose = 1).
   // ▄▄▄▄▄▄▄▄▄▄▄▄▄▄▄▄▄▄▄▄▄▄▄▄▄▄▄▄▄▄▄▄▄▄▄▄▄▄▄▄▄▄▄▄
   RUNG wire#powerrail
      I_Contact( #STATIC_DATA.CONFIG_FBK_CLOSED_EN )
      wire#w1
      Div(in1 := #wrkTimeFbkClosedDer, in2 := 100.0, out => #wrkReal)
      Mul(in1 := #wrkReal, in2 := #STATIC_DATA.TIME_CLOSING_MAX, out => #wrkReal)
      Sub(in1 := #STATIC_DATA.TIME_CLOSING_MAX, in2 := #wrkReal, out => #calClosedElapsedTime)
   END_RUNG
   RUNG wire#w1
      { S7_Templates := "SrcType := Real" } LE_Contact(in1 := #calClosedElapsedTime, in2 := #k_TIME_OP_MIN)
      Move(in := #k_TIME_OP_MIN, out1 => #calClosedElapsedTime)
   END_RUNG
   RUNG wire#w1
      Contact( #DYNAMIC_DATA.status_Closing )
      { S7_Templates := "SrcType := Real" } LE_Contact(in1 := #DYNAMIC_DATA.actual_Operating_Timer, in2 := #calClosedElapsedTime)
      S_Coil( #DYNAMIC_DATA."$derived_fbk_closed" )
   END_RUNG
   RUNG wire#powerrail
      Contact( #STATIC_DATA.CONFIG_FBK_CLOSED_EN )
      wire#w2
      R_Coil( #DYNAMIC_DATA."$derived_fbk_closed" )
   END_RUNG
   RUNG wire#powerrail
      Contact( #DYNAMIC_DATA."$ctrl_OpenClose" )
   END_RUNG wire#w2
   // the same network as SCL:
   #_w1 := NOT #STATIC_DATA.CONFIG_FBK_CLOSED_EN;
   IF #_w1 THEN
       #wrkReal := #wrkTimeFbkClosedDer / 100.0;
       #wrkReal := #wrkReal * #STATIC_DATA.TIME_CLOSING_MAX;
       #calClosedElapsedTime := #STATIC_DATA.TIME_CLOSING_MAX - #wrkReal;
   END_IF;
   IF #_w1 AND (#calClosedElapsedTime <= #k_TIME_OP_MIN) THEN
       #calClosedElapsedTime := #k_TIME_OP_MIN;
   END_IF;
   IF #_w1 AND #DYNAMIC_DATA.status_Closing AND (#DYNAMIC_DATA.actual_Operating_Timer <= #calClosedElapsedTime) THEN
       #DYNAMIC_DATA."$derived_fbk_closed" := TRUE;
   END_IF;
   IF #STATIC_DATA.CONFIG_FBK_CLOSED_EN OR #DYNAMIC_DATA."$ctrl_OpenClose" THEN
       #DYNAMIC_DATA."$derived_fbk_closed" := FALSE;
   END_IF;
END_REGION

REGION Network 17: Signal Conditioning — Simulation mode — Open signal
   // ▀▀▀▀▀▀▀▀▀▀▀▀▀▀▀▀▀▀▀▀▀▀▀▀▀▀▀▀▀▀▀▀▀▀▀▀▀▀▀▀▀▀▀▀
   // If simulation mode is active, the simulated open position signal is set as follows:
   // 
   //    •   mode_SimValue = 0 (no feedback), $sim_fbk_open = 0
   // 
   //    •   mode_SimValue = 1 (permanently open), $sim_fbk_open = 1
   // 
   //    •   mode_SimValue = 2 (permanently closed), $sim_fbk_open = 0
   // 
   //    •   mode_SimValue = 3 (follow demand), $sim_fbk_open = $ctrl_OpenClose
   //      with appropriate delay (the simulated position will activate when the
   //      operation timer counts down to a value less than or equal to K_TIME_SIM_MIN
   // 
   // If simulation mode is not active,  $sim_fbk_open = 0
   // ▄▄▄▄▄▄▄▄▄▄▄▄▄▄▄▄▄▄▄▄▄▄▄▄▄▄▄▄▄▄▄▄▄▄▄▄▄▄▄▄▄▄▄▄
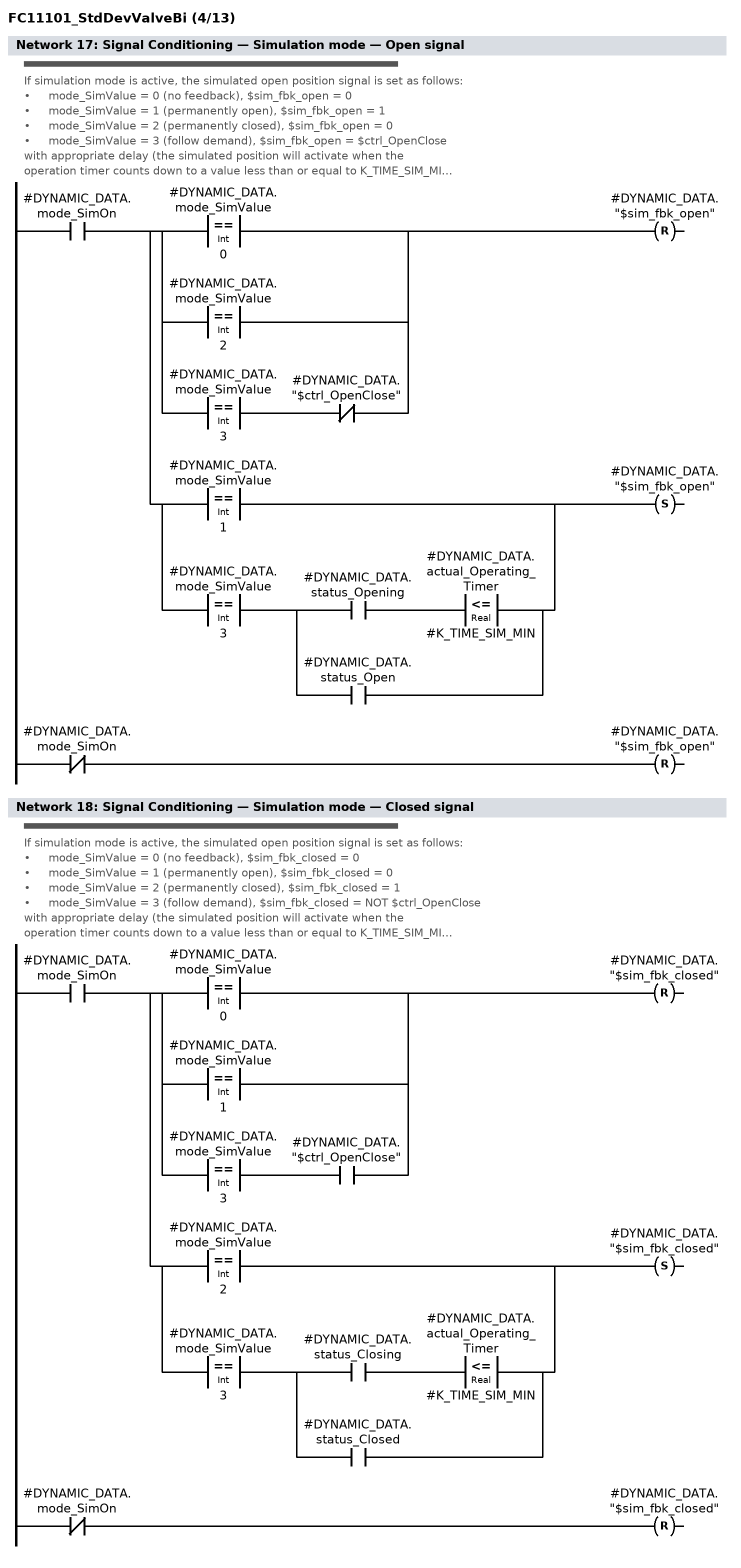
   RUNG wire#powerrail
      Contact( #DYNAMIC_DATA.mode_SimOn )
      wire#w1
      { S7_Templates := "SrcType := Int" } EQ_Contact(in1 := #DYNAMIC_DATA.mode_SimValue, in2 := 0)
      wire#w2
      R_Coil( #DYNAMIC_DATA."$sim_fbk_open" )
   END_RUNG
   RUNG wire#w1
      { S7_Templates := "SrcType := Int" } EQ_Contact(in1 := #DYNAMIC_DATA.mode_SimValue, in2 := 2)
   END_RUNG wire#w2
   RUNG wire#w1
      { S7_Templates := "SrcType := Int" } EQ_Contact(in1 := #DYNAMIC_DATA.mode_SimValue, in2 := 3)
      I_Contact( #DYNAMIC_DATA."$ctrl_OpenClose" )
   END_RUNG wire#w2
   RUNG wire#w1
      { S7_Templates := "SrcType := Int" } EQ_Contact(in1 := #DYNAMIC_DATA.mode_SimValue, in2 := 1)
      wire#w3
      S_Coil( #DYNAMIC_DATA."$sim_fbk_open" )
   END_RUNG
   RUNG wire#w1
      { S7_Templates := "SrcType := Int" } EQ_Contact(in1 := #DYNAMIC_DATA.mode_SimValue, in2 := 3)
      wire#w4
      Contact( #DYNAMIC_DATA.status_Opening )
      { S7_Templates := "SrcType := Real" } LE_Contact(in1 := #DYNAMIC_DATA.actual_Operating_Timer, in2 := #K_TIME_SIM_MIN)
   END_RUNG wire#w3
   RUNG wire#w4
      Contact( #DYNAMIC_DATA.status_Open )
   END_RUNG wire#w3
   RUNG wire#powerrail
      I_Contact( #DYNAMIC_DATA.mode_SimOn )
      R_Coil( #DYNAMIC_DATA."$sim_fbk_open" )
   END_RUNG
   // the same network as SCL:
   IF #DYNAMIC_DATA.mode_SimOn AND ((#DYNAMIC_DATA.mode_SimValue = 0) OR (#DYNAMIC_DATA.mode_SimValue = 2) OR ((#DYNAMIC_DATA.mode_SimValue = 3) AND NOT #DYNAMIC_DATA."$ctrl_OpenClose")) THEN
       #DYNAMIC_DATA."$sim_fbk_open" := FALSE;
   END_IF;
   IF #DYNAMIC_DATA.mode_SimOn AND ((#DYNAMIC_DATA.mode_SimValue = 1) OR ((#DYNAMIC_DATA.mode_SimValue = 3) AND ((#DYNAMIC_DATA.status_Opening AND (#DYNAMIC_DATA.actual_Operating_Timer <= #K_TIME_SIM_MIN)) OR #DYNAMIC_DATA.status_Open))) THEN
       #DYNAMIC_DATA."$sim_fbk_open" := TRUE;
   END_IF;
   IF NOT #DYNAMIC_DATA.mode_SimOn THEN #DYNAMIC_DATA."$sim_fbk_open" := FALSE; END_IF;
END_REGION

REGION Network 18: Signal Conditioning — Simulation mode — Closed signal
   // ▀▀▀▀▀▀▀▀▀▀▀▀▀▀▀▀▀▀▀▀▀▀▀▀▀▀▀▀▀▀▀▀▀▀▀▀▀▀▀▀▀▀▀▀
   // If simulation mode is active, the simulated open position signal is set as follows:
   // 
   //    •   mode_SimValue = 0 (no feedback), $sim_fbk_closed = 0
   // 
   //    •   mode_SimValue = 1 (permanently open), $sim_fbk_closed = 0
   // 
   //    •   mode_SimValue = 2 (permanently closed), $sim_fbk_closed = 1
   // 
   //    •   mode_SimValue = 3 (follow demand), $sim_fbk_closed = NOT $ctrl_OpenClose
   //      with appropriate delay (the simulated position will activate when the
   //      operation timer counts down to a value less than or equal to K_TIME_SIM_MIN
   // 
   // If simulation mode is not active,  $sim_fbk_closed = 0
   // ▄▄▄▄▄▄▄▄▄▄▄▄▄▄▄▄▄▄▄▄▄▄▄▄▄▄▄▄▄▄▄▄▄▄▄▄▄▄▄▄▄▄▄▄
   RUNG wire#powerrail
      Contact( #DYNAMIC_DATA.mode_SimOn )
      wire#w1
      { S7_Templates := "SrcType := Int" } EQ_Contact(in1 := #DYNAMIC_DATA.mode_SimValue, in2 := 0)
      wire#w2
      R_Coil( #DYNAMIC_DATA."$sim_fbk_closed" )
   END_RUNG
   RUNG wire#w1
      { S7_Templates := "SrcType := Int" } EQ_Contact(in1 := #DYNAMIC_DATA.mode_SimValue, in2 := 1)
   END_RUNG wire#w2
   RUNG wire#w1
      { S7_Templates := "SrcType := Int" } EQ_Contact(in1 := #DYNAMIC_DATA.mode_SimValue, in2 := 3)
      Contact( #DYNAMIC_DATA."$ctrl_OpenClose" )
   END_RUNG wire#w2
   RUNG wire#w1
      { S7_Templates := "SrcType := Int" } EQ_Contact(in1 := #DYNAMIC_DATA.mode_SimValue, in2 := 2)
      wire#w3
      S_Coil( #DYNAMIC_DATA."$sim_fbk_closed" )
   END_RUNG
   RUNG wire#w1
      { S7_Templates := "SrcType := Int" } EQ_Contact(in1 := #DYNAMIC_DATA.mode_SimValue, in2 := 3)
      wire#w4
      Contact( #DYNAMIC_DATA.status_Closing )
      { S7_Templates := "SrcType := Real" } LE_Contact(in1 := #DYNAMIC_DATA.actual_Operating_Timer, in2 := #K_TIME_SIM_MIN)
   END_RUNG wire#w3
   RUNG wire#w4
      Contact( #DYNAMIC_DATA.status_Closed )
   END_RUNG wire#w3
   RUNG wire#powerrail
      I_Contact( #DYNAMIC_DATA.mode_SimOn )
      R_Coil( #DYNAMIC_DATA."$sim_fbk_closed" )
   END_RUNG
   // the same network as SCL:
   IF #DYNAMIC_DATA.mode_SimOn AND ((#DYNAMIC_DATA.mode_SimValue = 0) OR (#DYNAMIC_DATA.mode_SimValue = 1) OR ((#DYNAMIC_DATA.mode_SimValue = 3) AND #DYNAMIC_DATA."$ctrl_OpenClose")) THEN
       #DYNAMIC_DATA."$sim_fbk_closed" := FALSE;
   END_IF;
   IF #DYNAMIC_DATA.mode_SimOn AND ((#DYNAMIC_DATA.mode_SimValue = 2) OR ((#DYNAMIC_DATA.mode_SimValue = 3) AND ((#DYNAMIC_DATA.status_Closing AND (#DYNAMIC_DATA.actual_Operating_Timer <= #K_TIME_SIM_MIN)) OR #DYNAMIC_DATA.status_Closed))) THEN
       #DYNAMIC_DATA."$sim_fbk_closed" := TRUE;
   END_IF;
   IF NOT #DYNAMIC_DATA.mode_SimOn THEN #DYNAMIC_DATA."$sim_fbk_closed" := FALSE; END_IF;
END_REGION

REGION Network 19: Signal conditioning — Determine valve OPEN position status
   // ▀▀▀▀▀▀▀▀▀▀▀▀▀▀▀▀▀▀▀▀▀▀▀▀▀▀▀▀▀▀▀▀▀▀▀▀▀▀▀▀▀▀▀▀
   // Generates a working open signal (wrkOpen), that is then used throughout the module as the 
   // definitive open position feedback signal.
   // 
   // The open signal will be either :
   // 
   //    1.  The same as the FBK_OPEN parameter if this is in use 
   //      (CONFIG_FBK_OPEN_EN = 1)
   // 
   //    2.  The internally derived open state (based on the requested state of the valve) if the 
   //      FBK_OPEN signal is NOT in use (CONFIG_FBK_OPEN_EN = 0)
   // 
   //    3.  The simulated state of the valve if simulation mode is active (mode_SimOn = 1)
   // 
   // If an actual open position signal is provided to the module via the FBK_OPEN parameter 
   // (i.e. if CONFIG_FBK_OPEN_EN = 1) then wrkOpen is set to match the FBK_OPEN signal 
   // (wrkOpen = FBK_OPEN).
   // 
   // If a derived open signal is to be used (i.e. if CONFIG_FBK_OPEN_EN = 0), then wrkOpen is set to 
   // match the internally derived $derived_fbk_open signal (wrkOpen = $derived_fbk_open). 
   // $derived_fbk_open is based on the requested state of the valve. 
   // 
   // Finally, if simulation mode is active (mode_SimOn = 1), then wrkOpen is set to match the internal 
   // simulation signal $sim_fbk_open signal (wrkOpen = $sim_fbk_open).. 
   // ▄▄▄▄▄▄▄▄▄▄▄▄▄▄▄▄▄▄▄▄▄▄▄▄▄▄▄▄▄▄▄▄▄▄▄▄▄▄▄▄▄▄▄▄
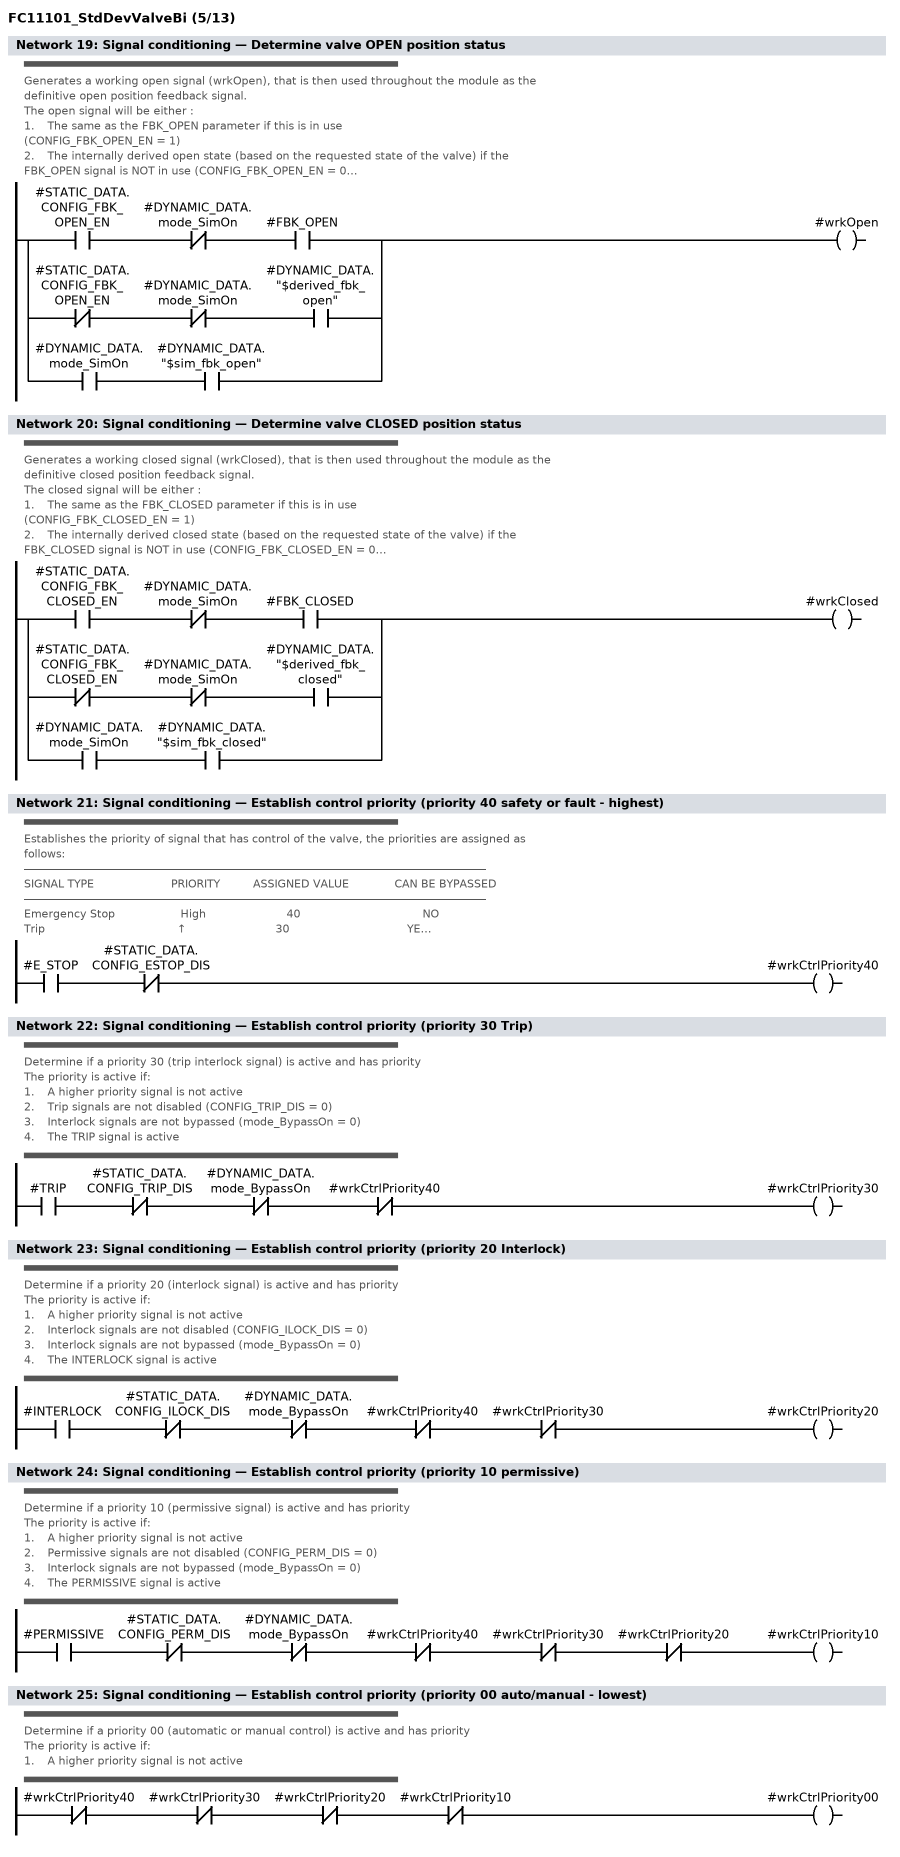
   RUNG wire#powerrail
      Contact( #STATIC_DATA.CONFIG_FBK_OPEN_EN )
      I_Contact( #DYNAMIC_DATA.mode_SimOn )
      Contact( #FBK_OPEN )
      wire#w1
      Coil( #wrkOpen )
   END_RUNG
   RUNG wire#powerrail
      I_Contact( #STATIC_DATA.CONFIG_FBK_OPEN_EN )
      I_Contact( #DYNAMIC_DATA.mode_SimOn )
      Contact( #DYNAMIC_DATA."$derived_fbk_open" )
   END_RUNG wire#w1
   RUNG wire#powerrail
      Contact( #DYNAMIC_DATA.mode_SimOn )
      Contact( #DYNAMIC_DATA."$sim_fbk_open" )
   END_RUNG wire#w1
   // the same network as SCL:
   #wrkOpen := (#STATIC_DATA.CONFIG_FBK_OPEN_EN AND NOT #DYNAMIC_DATA.mode_SimOn AND #FBK_OPEN) OR (NOT #STATIC_DATA.CONFIG_FBK_OPEN_EN AND NOT #DYNAMIC_DATA.mode_SimOn AND #DYNAMIC_DATA."$derived_fbk_open") OR (#DYNAMIC_DATA.mode_SimOn AND #DYNAMIC_DATA."$sim_fbk_open");
END_REGION

REGION Network 20: Signal conditioning — Determine valve CLOSED position status
   // ▀▀▀▀▀▀▀▀▀▀▀▀▀▀▀▀▀▀▀▀▀▀▀▀▀▀▀▀▀▀▀▀▀▀▀▀▀▀▀▀▀▀▀▀
   // Generates a working closed signal (wrkClosed), that is then used throughout the module as the 
   // definitive closed position feedback signal.
   // 
   // The closed signal will be either :
   // 
   //    1.  The same as the FBK_CLOSED parameter if this is in use 
   //      (CONFIG_FBK_CLOSED_EN = 1)
   // 
   //    2.  The internally derived closed state (based on the requested state of the valve) if the 
   //      FBK_CLOSED signal is NOT in use (CONFIG_FBK_CLOSED_EN = 0)
   // 
   //    3.  The simulated state of the valve if simulation mode is active (mode_SimOn = 1)
   // 
   // If an actual closed position signal is provided to the module via the FBK_CLOSED parameter 
   // (i.e. if CONFIG_FBK_CLOSED_EN = 1) then wrkClosed is set to match the FBK_CLOSED signal 
   // wrkClosed = FBK_CLOSED).
   // 
   // If a derived closed signal is to be used (i.e. if CONFIG_FBK_CLOSED_EN = 0), then wrkClosed is 
   // set to match the internally derived $derived_fbk_closed signal 
   // (wrkClosed = $derived_fbk_closed). $derived_fbk_closed is based on the requested state of 
   // the valve.
   // 
   // Finally, if simulation mode is active (mode_SimOn = 1), then wrkClosed is set to match the 
   // internal simulation signal $sim_fbk_closed signal (wrkClosed = $sim_fbk_closed). 
   // ▄▄▄▄▄▄▄▄▄▄▄▄▄▄▄▄▄▄▄▄▄▄▄▄▄▄▄▄▄▄▄▄▄▄▄▄▄▄▄▄▄▄▄▄
   RUNG wire#powerrail
      Contact( #STATIC_DATA.CONFIG_FBK_CLOSED_EN )
      I_Contact( #DYNAMIC_DATA.mode_SimOn )
      Contact( #FBK_CLOSED )
      wire#w1
      Coil( #wrkClosed )
   END_RUNG
   RUNG wire#powerrail
      I_Contact( #STATIC_DATA.CONFIG_FBK_CLOSED_EN )
      I_Contact( #DYNAMIC_DATA.mode_SimOn )
      Contact( #DYNAMIC_DATA."$derived_fbk_closed" )
   END_RUNG wire#w1
   RUNG wire#powerrail
      Contact( #DYNAMIC_DATA.mode_SimOn )
      Contact( #DYNAMIC_DATA."$sim_fbk_closed" )
   END_RUNG wire#w1
   // the same network as SCL:
   #wrkClosed := (#STATIC_DATA.CONFIG_FBK_CLOSED_EN AND NOT #DYNAMIC_DATA.mode_SimOn AND #FBK_CLOSED) OR (NOT #STATIC_DATA.CONFIG_FBK_CLOSED_EN AND NOT #DYNAMIC_DATA.mode_SimOn AND #DYNAMIC_DATA."$derived_fbk_closed") OR (#DYNAMIC_DATA.mode_SimOn AND #DYNAMIC_DATA."$sim_fbk_closed");
END_REGION

REGION Network 21: Signal conditioning — Establish control priority (priority 40 safety or fault - highest)
   // ▀▀▀▀▀▀▀▀▀▀▀▀▀▀▀▀▀▀▀▀▀▀▀▀▀▀▀▀▀▀▀▀▀▀▀▀▀▀▀▀▀▀▀▀
   // Establishes the priority of signal that has control of the valve, the priorities are assigned as 
   // follows:
   // 
   //  ――――――――――――――――――――――――――――――――――――――――――
   //  SIGNAL TYPE       PRIORITY   ASSIGNED VALUE       CAN BE BYPASSED
   //  ――――――――――――――――――――――――――――――――――――――――――
   //  Emergency Stop        High        40                NO
   //  Trip            ↑           30             YES
   //  Interlock            ↑           20             YES
   //  Permissive          ↑           10             YES
   //  Auto/manual control    Low         00                NO
   //  ――――――――――――――――――――――――――――――――――――――――――
   //  High priority signal take precedence over lower priority signals.
   // 
   // Determine a priority 40 (valve safety (or fault) condition is active)
   // 
   // The priority is active if:
   // 
   //    1.  Safety signals are not disabled (CONFIG_ESTOP_DIS = 0)
   // 
   //    2.  The E_STOP signal is active
   // ▄▄▄▄▄▄▄▄▄▄▄▄▄▄▄▄▄▄▄▄▄▄▄▄▄▄▄▄▄▄▄▄▄▄▄▄▄▄▄▄▄▄▄▄
   RUNG wire#powerrail
      Contact( #E_STOP )
      I_Contact( #STATIC_DATA.CONFIG_ESTOP_DIS )
      Coil( #wrkCtrlPriority40 )
   END_RUNG
   // the same network as SCL:
   #wrkCtrlPriority40 := #E_STOP AND NOT #STATIC_DATA.CONFIG_ESTOP_DIS;
END_REGION

REGION Network 22: Signal conditioning — Establish control priority (priority 30 Trip)
   // ▀▀▀▀▀▀▀▀▀▀▀▀▀▀▀▀▀▀▀▀▀▀▀▀▀▀▀▀▀▀▀▀▀▀▀▀▀▀▀▀▀▀▀▀
   // Determine if a priority 30 (trip interlock signal) is active and has priority
   // 
   // The priority is active if:
   // 
   //    1.  A higher priority signal is not active
   // 
   //    2.  Trip signals are not disabled (CONFIG_TRIP_DIS = 0)
   // 
   //    3.  Interlock signals are not bypassed (mode_BypassOn = 0)
   // 
   //    4.  The TRIP signal is active
   // ▄▄▄▄▄▄▄▄▄▄▄▄▄▄▄▄▄▄▄▄▄▄▄▄▄▄▄▄▄▄▄▄▄▄▄▄▄▄▄▄▄▄▄▄
   RUNG wire#powerrail
      Contact( #TRIP )
      I_Contact( #STATIC_DATA.CONFIG_TRIP_DIS )
      I_Contact( #DYNAMIC_DATA.mode_BypassOn )
      I_Contact( #wrkCtrlPriority40 )
      Coil( #wrkCtrlPriority30 )
   END_RUNG
   // the same network as SCL:
   #wrkCtrlPriority30 := #TRIP AND NOT #STATIC_DATA.CONFIG_TRIP_DIS AND NOT #DYNAMIC_DATA.mode_BypassOn AND NOT #wrkCtrlPriority40;
END_REGION

REGION Network 23: Signal conditioning — Establish control priority (priority 20 Interlock)
   // ▀▀▀▀▀▀▀▀▀▀▀▀▀▀▀▀▀▀▀▀▀▀▀▀▀▀▀▀▀▀▀▀▀▀▀▀▀▀▀▀▀▀▀▀
   // Determine if a priority 20 (interlock signal) is active and has priority
   // 
   // The priority is active if:
   // 
   //    1.  A higher priority signal is not active
   // 
   //    2.  Interlock signals are not disabled (CONFIG_ILOCK_DIS = 0)
   // 
   //    3.  Interlock signals are not bypassed (mode_BypassOn = 0)
   // 
   //    4.  The INTERLOCK signal is active
   // ▄▄▄▄▄▄▄▄▄▄▄▄▄▄▄▄▄▄▄▄▄▄▄▄▄▄▄▄▄▄▄▄▄▄▄▄▄▄▄▄▄▄▄▄
   RUNG wire#powerrail
      Contact( #INTERLOCK )
      I_Contact( #STATIC_DATA.CONFIG_ILOCK_DIS )
      I_Contact( #DYNAMIC_DATA.mode_BypassOn )
      I_Contact( #wrkCtrlPriority40 )
      I_Contact( #wrkCtrlPriority30 )
      Coil( #wrkCtrlPriority20 )
   END_RUNG
   // the same network as SCL:
   #wrkCtrlPriority20 := #INTERLOCK AND NOT #STATIC_DATA.CONFIG_ILOCK_DIS AND NOT #DYNAMIC_DATA.mode_BypassOn AND NOT #wrkCtrlPriority40 AND NOT #wrkCtrlPriority30;
END_REGION

REGION Network 24: Signal conditioning — Establish control priority (priority 10 permissive)
   // ▀▀▀▀▀▀▀▀▀▀▀▀▀▀▀▀▀▀▀▀▀▀▀▀▀▀▀▀▀▀▀▀▀▀▀▀▀▀▀▀▀▀▀▀
   // Determine if a priority 10 (permissive signal) is active and has priority
   // 
   // The priority is active if:
   // 
   //    1.  A higher priority signal is not active
   // 
   //    2.  Permissive signals are not disabled (CONFIG_PERM_DIS = 0)
   // 
   //    3.  Interlock signals are not bypassed (mode_BypassOn = 0)
   // 
   //    4.  The PERMISSIVE signal is active
   // ▄▄▄▄▄▄▄▄▄▄▄▄▄▄▄▄▄▄▄▄▄▄▄▄▄▄▄▄▄▄▄▄▄▄▄▄▄▄▄▄▄▄▄▄
   RUNG wire#powerrail
      Contact( #PERMISSIVE )
      I_Contact( #STATIC_DATA.CONFIG_PERM_DIS )
      I_Contact( #DYNAMIC_DATA.mode_BypassOn )
      I_Contact( #wrkCtrlPriority40 )
      I_Contact( #wrkCtrlPriority30 )
      I_Contact( #wrkCtrlPriority20 )
      Coil( #wrkCtrlPriority10 )
   END_RUNG
   // the same network as SCL:
   #wrkCtrlPriority10 := #PERMISSIVE AND NOT #STATIC_DATA.CONFIG_PERM_DIS AND NOT #DYNAMIC_DATA.mode_BypassOn AND NOT #wrkCtrlPriority40 AND NOT #wrkCtrlPriority30 AND NOT #wrkCtrlPriority20;
END_REGION

REGION Network 25: Signal conditioning — Establish control priority (priority 00 auto/manual - lowest)
   // ▀▀▀▀▀▀▀▀▀▀▀▀▀▀▀▀▀▀▀▀▀▀▀▀▀▀▀▀▀▀▀▀▀▀▀▀▀▀▀▀▀▀▀▀
   // Determine if a priority 00 (automatic or manual control) is active and has priority
   // 
   // The priority is active if:
   // 
   //    1.  A higher priority signal is not active
   // ▄▄▄▄▄▄▄▄▄▄▄▄▄▄▄▄▄▄▄▄▄▄▄▄▄▄▄▄▄▄▄▄▄▄▄▄▄▄▄▄▄▄▄▄
   RUNG wire#powerrail
      I_Contact( #wrkCtrlPriority40 )
      I_Contact( #wrkCtrlPriority30 )
      I_Contact( #wrkCtrlPriority20 )
      I_Contact( #wrkCtrlPriority10 )
      Coil( #wrkCtrlPriority00 )
   END_RUNG
   // the same network as SCL:
   #wrkCtrlPriority00 := NOT #wrkCtrlPriority40 AND NOT #wrkCtrlPriority30 AND NOT #wrkCtrlPriority20 AND NOT #wrkCtrlPriority10;
END_REGION

